// TIA Portal project "OI455" (V15.1)

(* hardware
DEVICE "ET 200SP station_1"  ET 200SP-Station
   slot 0: "Rack_0"  Rack  6ES5 710-8MAx1
   slot 1: "PLC_1"  CPU 1512SP-1 PN  6ES7 512-1DK01-0AB0  V2.6
   slot 2: "CM PtP_1"  CM PtP  6ES7 137-6AA00-0BA0  V1.0
      slot 1: "CM PtP_1"  CM PtP Sub
   slot 3: "CM PtP_2"  CM PtP  6ES7 137-6AA00-0BA0  V1.0
      slot 1: "CM PtP_2"  CM PtP Sub
   slot 4: "DI 8x24VDC BA_1"  DI 8x24VDC BA  6ES7 131-6BF01-0AA0  V0.0
      slot 1: "DI 8x24VDC BA_1"  DI 8x24VDC BA
   slot 5: "DI 8x24VDC BA_2"  DI 8x24VDC BA  6ES7 131-6BF01-0AA0  V0.0
      slot 1: "DI 8x24VDC BA_2"  DI 8x24VDC BA
   slot 6: "DI 8x24VDC BA_3"  DI 8x24VDC BA  6ES7 131-6BF01-0AA0  V0.0
      slot 1: "DI 8x24VDC BA_3"  DI 8x24VDC BA
   slot 7: "DQ 8x24VDC/0.5A BA_1"  DQ 8x24VDC/0.5A BA  6ES7 132-6BF01-0AA0  V0.0
      slot 1: "DQ 8x24VDC/0.5A BA_1"  DQ 8x24VDC/0.5A BA
   slot 8: "DQ 8x24VDC/0.5A BA_2"  DQ 8x24VDC/0.5A BA  6ES7 132-6BF01-0AA0  V0.0
      slot 1: "DQ 8x24VDC/0.5A BA_2"  DQ 8x24VDC/0.5A BA
   slot 9: "AI 8xI 2-,4-wire BA_1"  AI 8xI 2-,4-wire BA  6ES7 134-6GF00-0AA1  V1.0
      slot 1: "AI 8xI 2-,4-wire BA_1"  AI 8xI 2-,4-wire BA
   slot 10: "AI 8xI 2-,4-wire BA_2"  AI 8xI 2-,4-wire BA  6ES7 134-6GF00-0AA1  V1.0
      slot 1: "AI 8xI 2-,4-wire BA_2"  AI 8xI 2-,4-wire BA
   slot 11: "Server module_1"  Server module  6ES7 193-6PA00-0AA0  V1.1
      slot 1: "Server module_1"  Server module
   slot 127: "BA 2xRJ45"  BA 2xRJ45  6ES7 193-6AR00-0AA0  V0.0
      slot 32769: "Port_1"  6ES7 193-6AR00-0AA0
      slot 32770: "Port_2"  6ES7 193-6AR00-0AA0
*)

// ===== PLC "PLC_1"  CPU 1512SP-1 PN =====

VAR_GLOBAL   // PLC tag table "Default tag table"
   "AI2_Ch0" AT %IW35 : Word;
   "AI2_Ch1" AT %IW37 : Word;
   "AI2_Ch2" AT %IW39 : Word;
   "AI2_Ch3" AT %IW41 : Word;
   "AI2_Ch4" AT %IW43 : Word;
   "AI2_Ch5" AT %IW45 : Word;
   "AI2_Ch6" AT %IW47 : Word;
   "AI2_Ch7" AT %IW49 : Word;
   "AI1_Ch0" AT %IW19 : Word;
   "AI1_Ch1" AT %IW21 : Word;
   "AI1_Ch2" AT %IW23 : Word;
   "AI1_Ch3" AT %IW25 : Word;
   "AI1_Ch4" AT %IW27 : Word;
   "AI1_Ch5" AT %IW29 : Word;
   "AI1_Ch6" AT %IW31 : Word;
   "AI1_Ch7" AT %IW33 : Word;
   "DI1_In" AT %IB16 : Byte;
   "DI2_In" AT %IB17 : Byte;
   "DI3_In" AT %IB18 : Byte;
   "DO1_Out" AT %QB0 : Byte;
   "DO2_Out" AT %QB1 : Byte;
   "System_Byte" AT %MB1 : Byte;
   "FirstScan" AT %M1.0 : Bool;
   "DiagStatusUpdate" AT %M1.1 : Bool;
   "AlwaysTRUE" AT %M1.2 : Bool;
   "AlwaysFALSE" AT %M1.3 : Bool;
   "Clock_Byte" AT %MB0 : Byte;
   "Clock_10Hz" AT %M0.0 : Bool;
   "Clock_5Hz" AT %M0.1 : Bool;
   "Clock_2.5Hz" AT %M0.2 : Bool;
   "Clock_2Hz" AT %M0.3 : Bool;
   "Clock_1.25Hz" AT %M0.4 : Bool;
   "Clock_1Hz" AT %M0.5 : Bool;
   "Clock_0.625Hz" AT %M0.6 : Bool;
   "Clock_0.5Hz" AT %M0.7 : Bool;
   "ReqUVP" AT %M20.0 : Bool;
   "PrevState" AT %MW30 : Int;
   "HS600_active" AT %M20.1 : Bool;
   "Alarm_protect_XV100" AT %M20.2 : Bool;
   "Alarm_protect_XV100_prev" AT %M20.3 : Bool;
   "Alarm_Gas" AT %M20.4 : Bool;
   "Alarm_Gas_prev" AT %M20.5 : Bool;
   "Head_cmd_on_prev" AT %M20.6 : Bool;
   "Head_cmd_off_prev" AT %M20.7 : Bool;
   "Power_cmd_on_prev" AT %M21.0 : Bool;
   "Power_cmd_off_prev" AT %M21.1 : Bool;
   "CommandHMI_Spark_prev" AT %M21.2 : Bool;
   "Power_reset_prev" AT %M21.3 : Bool;
   "Head_reset_prev" AT %M21.4 : Bool;
END_VAR

TYPE "dt_AI"
   STRUCT
      Acp : DInt;   // Actual ADC code
      State : Word;
      Value : Real;   // Actual value (eng.units)
      Value_LastScan : Real;   // Last scan value
      K_filtr : Real := 0.0;   // Filter quoficient ( enable if K_filtr>0 )
      Circuit : Real;   // Actual current(mA)
      Voltage : Real;   // Actual vlotage (V)
      Resistance : Real;   // Input resistance (for voltage inputs)
      Scal_Max_Eu : Real := 100.0;   // Max scale value (eng.units)
      Scal_Min_Eu : Real := 0.0;   // Min scale value (eng.units)
      HH_Lim : Real := 100.0;   // HiHi alarm SP (eng.units)
      H_Lim : Real := 95.0;   // Hi warning SP (eng.units)
      L_Lim : Real := 5.0;   // Low warning SP (eng.units)
      LL_Lim : Real := 0.0;   // LowLow alarm SP (eng.units)
      HH_DeadBand : Real;   // HiHi alarm deadband
      H_DeadBand : Real;   // Hi warning deadband
      L_DeadBand : Real;   // Low warning deadband
      LL_DeadBand : Real;   // LowLow alarm deadband
      HH_Delay : Time;   // HiHi alarm SP delay
      H_Delay : Time;   // Hi warning SP delay
      L_Delay : Time;   // Low warning SP delay
      LL_Delay : Time;   // LowLow alarm SP delay
      Sim_Value : Real;   // Simulate value (eng.units)
      Sim_En : Bool := FALSE;   // Enable simulate mode
      Scal_Max_Upper : Bool;   // Flag Hi scale overflow
      Scal_Min_Under : Bool;   // Flag Low scale underflow
      Scale_0_20mA : Bool := FALSE;   // True - 0-20 mA, False - 4-20 mA
      Input_4mA_on_0_20mA : Bool := TRUE;   // True - 4-20mA sensor on 0-20mA current input
      VoltageInputType : Bool := FALSE;   // True -- voltage inpit, False - circuit input
      HH_Alarm : Bool;   // HiHi alarm flag
      H_Alarm : Bool;   // Hi warning flag
      L_Alarm : Bool;   // Low warning flag
      LL_Alarm : Bool;   // LowLow alarm flag
      HH_Alarm_En : Bool := TRUE;   // Enable HiHi alarm
      H_Alarm_En : Bool := FALSE;   // Enable Hi warning
      L_Alarm_En : Bool := FALSE;   // Enable Low warning
      LL_Alarm_En : Bool := TRUE;   // Enable LowLow alarm
      Short_Circuit : Bool;   // Shortcut flag
      Break : Bool;   // Breakoff flag
      Chan_Fail : Bool;   // Channel fault flag
      HH_Alarm_Logic : Bool;   // HiHi alarm for logic
      H_Alarm_Logic : Bool;   // Hi warning for logic
      L_Alarm_Logic : Bool;   // Low warning for logic
      LL_Alarm_Logic : Bool;   // LowLow alarm for logic
      Chan_Fail_Logic : Bool;   // Channel fault for logic
      Mask_mode : Bool;
      Test_mode : Bool;
      Ack_HH : Bool;
      Ack_H : Bool;
      Ack_L : Bool;
      Ack_LL : Bool;
      State_color : Byte;   // for HMI
      Ack_Alarm : Byte;   // for HMI
      Ack_Warning : Byte;   // for HMI
   END_STRUCT;
END_TYPE

TYPE "dt_DO"
   STRUCT
      Data_to_out : Word;
      Pins : Array[0..15] of Bool;
      UsePinsAsInput : Bool;
      Invert_En : Word;
      Output_En : Word;
      Sim_En : Word;
      Sim_Value : Word;
      Value : Word;
   END_STRUCT;
END_TYPE

TYPE "UVP_Param"
   STRUCT
      Connect_ID : UInt;
      IP_OCTET1 : UInt;
      IP_OCTET2 : UInt;
      IP_OCTET3 : UInt;
      IP_OCTET4 : UInt;
      IP_PORT : UInt;
   END_STRUCT;
END_TYPE

TYPE "Setpoints_v2"
   STRUCT
      UVPTimeCorrection : Real;
      reserv_4 : Real;
      reserv_5 : Real;
      reserv_6 : Real;
      Temp_L1_Press : Real;   // нижняя предупредительная уставка расхода газа на линии 2
      Temp_L1_Abs_Press : Real;
      Temp_L2_Press : Real;
      Temp_L2_Abs_Press : Real;
      Temp_L3_Press : Real;
      Temp_L3_Abs_Press : Real;
      Temp_L4_Press : Real;
      Temp_L4_Abs_Press : Real;
   END_STRUCT;
END_TYPE

TYPE "MeasuredUVP"
   STRUCT
      UVP_Press : Real;   // Избыточное давление, Па
      UVP_Abs_press : Real;   // Абсолютное давление, Па
      UVP_Temp : Real;   // Температура газа, С
      UVP_Ent : Real;   // Энтальпия, Дж/кг
      UVP_mass_flow : Real;   // Масовый расход, кг/сек
      UVP_Mass : Real;   // Масса, кг
      UVP_Vol_work : Real;   // Объем в р.у., м3
      UVP_Vol_norm : Real;   // Объем в ст.у., нм3
      UVP_T_power : Real;   // Тепловая мощность, Вт
      UVP_T_energ : Real;   // Тепловая энергия, Дж
      UVP_Time : DInt;   // Время штатной работы, сек
      UVP_TimeEr : DInt;   // Время нештатных ситуаций, сек
      UVP_Param_m_flow : Real;   // Параметр датчика расхода/количества, кг/сек
      UVP_Param_vol_flow_work : Real;   // Параметр датчика расхода/количества (в р.у.), м3/сек
      UVP_Param_vol_flow_norm : Real;   // Параметр датчика расхода/количества (в ст.у.), нм3/сек
      UVP_Param_mass : Real;   // Параметр датчика расхода/количества (масса), кг
      UVP_Param_vol : Real;   // Параметр датчика расхода/количества (объём в р.у.), м3
      UVP_NotUsed : Real;   // Резерв
      UVP_Density_norm : Real;   // Текущее значение плотности среды в ст.у, кг/м3
      UVP_Density_work : Real;   // Текущее значение плотности среды в р.у, кг/м3
      UVP_dP : Real;   // Перепад давления для трубопроводов на СУ, Па
      UVP_vol_flow_norm : Real;   // Объемный расход в ст.у. нм3/с
      UVP_vol_flow_work : Real;   // Объемный расход в р.у. нм3/с
   END_STRUCT;
END_TYPE

TYPE "CumulativeUVP"
   STRUCT
      UVP_Mass_prev2h : Real;   // Масса за предыд. час/2 часа, кг
      UVP_Vol_work_prev2h : Real;   // Объём в р.у за предыд. час/2 часа, м3
      UVP_Vol_norm_prev2h : Real;   // Объём в ст.у за предыд. час/2 часа, нм3
      UVP_Param_m_flow_prev2h : Real;   // Параметр датчика расхода/количества за предыд. час/2 часа, кг
      UVP_Param_vol_flow_work_prev2h : Real;   // Параметр датчика расхода/количества (объём в р.у.) за предыд. час/2 часа, м3
      UVP_Mass_cumul2h : Real;   // Масса на конец предыд. час/2 часа, кг
      UVP_Vol_work_cumul2h : Real;   // Объём на конец р.у за предыд. час/2 часа, м3
      UVP_Vol_norm_cumul2h : Real;   // Объём на конец ст.у за предыд. час/2 часа, нм3
      UVP_Param_m_flow_cumul2h : Real;   // Параметр датчика расхода/количества на конец предыд. час/2 часа, кг
      UVP_Param_vol_flow_work_cumul2h : Real;   // Параметр датчика расхода/количества (объём в р.у.) на конец предыд. час/2 часа, м3
      UVP_Mass_prevDay : Real;   // Масса за предыд. сутки, кг
      UVP_Vol_work_prevDay : Real;   // Объём в р.у за предыд. сутки, м3
      UVP_Vol_norm_prevDay : Real;   // Объём в ст.у за предыд. сутки, нм3
      UVP_Param_m_flow_prevDay : Real;   // Параметр датчика расхода/количества за предыд. сутки, кг
      UVP_Param_vol_flow_work_prevDay : Real;   // Параметр датчика расхода/количества (объём в р.у.) за предыд. сутки, м3
      UVP_Mass_cumulDay : Real;   // Масса на конец предыд. суток, кг
      UVP_Vol_work_cumulDay : Real;   // Объём на конец р.у за предыд. суток, м3
      UVP_Vol_norm_cumulDay : Real;   // Объём на конец ст.у за предыд. суток, нм3
      UVP_Param_m_flow_cumulDay : Real;   // Параметр датчика расхода/количества на конец предыд. суток, кг
      UVP_Param_vol_flow_work_cumulDay : Real;   // Параметр датчика расхода/количества (объём в р.у.) на конец предыд. суток, м3
   END_STRUCT;
END_TYPE

TYPE "Commands_v2"
   STRUCT
      Set_IP_UVP1 : Bool;   // Изменить IP адрес УВП1
      Set_IP_UVP2 : Bool;   // Изменить IP адрес УВП2
      UVP_MR113_Read : Bool;   // Прочитать компонентный состав из УВП 1
      UVP_MR113_Write : Bool;   // Записать компонентный состав в УВП 1
      UVP2_MR113_Read : Bool;   // Прочитать компонентный состав из УВП 2
      UVP2_MR113_Write : Bool;   // Записать компонентный состав в УВП 2
      UVPArchReadStart : Bool;   // команда на чтение архивной записи
   END_STRUCT;
END_TYPE

TYPE "DateTimeUVP"
   STRUCT
      Day : Int;
      Month : Int;
      Year : Int;
      Hour : Int;
      Minute : Int;
      Second : Int;
   END_STRUCT;
END_TYPE

TYPE "MR113_03_Gas_UVP"
   STRUCT
      CH4 : Real;   // Концентрация CH4 метан (мольные доли либо массовый %)
      C2H6 : Real;   // Концентрация C2H6 этан (мольные доли либо массовый %)
      C3H8 : Real;   // Концентрация C3H8 пропан (мольные доли либо массовый %)
      nC4H10 : Real;   // Концентрация н-C4H10 н-бутан (мольные доли либо массовый %)
      iC4H10 : Real;   // Концентрация и-C4H10 и-бутан (мольные доли либо массовый %)
      nC5H12 : Real;   // Концентрация н-C5H12 н-пептан (мольные доли либо массовый %)
      N2 : Real;   // Концентрация N2 азот (мольные доли либо массовый %)
      CO2 : Real;   // Концентрация CO2 углекислота (мольные доли либо массовый %)
      H2O : Real;   // Концентрация H2O вода (мольные доли либо массовый %)
      H2S : Real;   // Концентрация H2S сероводород (мольные доли либо массовый %)
      C6H14 : Real;   // Концентрация C6H14 гексан (мольные доли либо массовый %)
      C7H16 : Real;   // Концентрация C7H16 гептан (мольные доли либо массовый %)
      O2 : Real;   // Концентрация O2 кислород (мольные доли либо массовый %)
      iC5H12 : Real;   // Концентрация и-C5H12 и-пептан (мольные доли либо массовый %)
      Humidity : Real;   // Влажность (абсолютное значение в г/м3 либо относительная концентрация)
   END_STRUCT;
END_TYPE

TYPE "Measured"
   STRUCT
      UVP1_L1_Archive_AbsPresAve : Real;   // Архивное давление, МПа (среднее за период) - УВП1 линия1
      UVP1_L1_Archive_AbsTempAve : Real;   // Архивная температура, С (средняя за период) - УВП1 линия1
      UVP1_L1_Archive_FlowWorkPeriod : Real := 0.0;   // Архивный расход за период (р.у.), м3 - УВП1 линия1
      UVP1_L1_Archive_FlowNormPeriod : Real := 0.0;   // Архивный расход за период (с.у.), нм3 - УВП1 линия1
      UVP1_L1_Archive_StableWorkTime : Real := 0.0;   // Время штатной работы, часов - УВП1 линия1
      reserv : Real := 0.0;   // резерв
      UVP1_L2_Archive_AbsPresAve : Real := 0.0;   // Архивное давление, МПа (среднее за период) - УВП1 линия2
      UVP1_L2_Archive_AbsTempAve : Real := 0.0;   // Архивная температура, С (средняя за период) - УВП1 линия2
      UVP1_L2_Archive_FlowWorkPeriod : Real := 0.0;   // Архивный расход за период (р.у.), м3 - УВП1 линия2
      UVP1_L2_Archive_FlowNormPeriod : Real := 0.0;   // Архивный расход за период (с.у.), нм3 - УВП1 линия2
      UVP1_L2_Archive_StableWorkTime : Real := 0.0;   // Время штатной работы, часов - УВП1 линия2
      reserv_6 : Real := 0.0;   // резерв
      UVP1_L3_Archive_AbsPresAve : Real := 0.0;   // Архивное давление, МПа (среднее за период) - УВП1 линия3
      UVP1_L3_Archive_AbsTempAve : Real := 0.0;   // Архивная температура, С (средняя за период) - УВП1 линия3
      UVP1_L3_Archive_FlowWorkPeriod : Real := 0.0;   // Архивный расход за период (р.у.), м3 - УВП1 линия3
      UVP1_L3_Archive_FlowNormPeriod : Real := 0.0;   // Архивный расход за период (с.у.), нм3 - УВП1 линия3
      UVP1_L3_Archive_StableWorkTime : Real := 0.0;   // Время штатной работы, часов - УВП1 линия3
      reserv_12 : Real := 0.0;   // резерв
      UVP1_L4_Archive_AbsPresAve : Real;   // Архивное давление, МПа (среднее за период) - УВП1 линия4
      UVP1_L4_Archive_AbsTempAve : Real;   // Архивная температура, С (средняя за период) - УВП1 линия4
      UVP1_L4_Archive_FlowWorkPeriod : Real;   // Архивный расход за период (р.у.), м3 - УВП1 линия4
      UVP1_L4_Archive_FlowNormPeriod : Real;   // Архивный расход за период (с.у.), нм3 - УВП1 линия4
      UVP1_L4_Archive_StableWorkTime : Real;   // Время штатной работы, часов - УВП1 линия4
      reserv_18 : Real;   // резерв
      UVP2_L1_Archive_AbsPresAve : Real;   // Архивное давление, МПа (среднее за период) - УВП1 линия1
      UVP2_L1_Archive_AbsTempAve : Real;   // Архивная температура, С (средняя за период) - УВП2 линия1
      UVP2_L1_Archive_FlowWorkPeriod : Real := 0.0;   // Архивный расход за период (р.у.), м3 - УВП2 линия1
      UVP2_L1_Archive_FlowNormPeriod : Real := 0.0;   // Архивный расход за период (с.у.), нм3 - УВП2 линия1
      UVP2_L1_Archive_StableWorkTime : Real := 0.0;   // Время штатной работы, часов - УВП2 линия1
      reserv_1 : Real := 0.0;   // резерв
      UVP2_L2_Archive_AbsPresAve : Real := 0.0;   // Архивное давление, МПа (среднее за период) - УВП2 линия2
      UVP2_L2_Archive_AbsTempAve : Real := 0.0;   // Архивная температура, С (средняя за период) - УВП2 линия2
      UVP2_L2_Archive_FlowWorkPeriod : Real := 0.0;   // Архивный расход за период (р.у.), м3 - УВП2 линия2
      UVP2_L2_Archive_FlowNormPeriod : Real := 0.0;   // Архивный расход за период (с.у.), нм3 - УВП2 линия2
      UVP2_L2_Archive_StableWorkTime : Real := 0.0;   // Время штатной работы, часов - УВП2 линия2
      reserv_7 : Real := 0.0;   // резерв
      reserv_19 : Real;   // резерв
   END_STRUCT;
END_TYPE

TYPE "MR113_03_Gas_UVP_Int"
   STRUCT
      Concentration : Int;
      Water : Int;
   END_STRUCT;
END_TYPE

TYPE "UVP_ArchiveResult"
   STRUCT
      UVP1_Archive_RequestStatus : Int;   // Статус чтения архива (для первого клиента): 0 - нет данных, 1 - идёт сбор, 2 - данные готовы, 3..7 - ошибки
      UVP2_Archive_RequestStatus : Int;   // Статус чтения архива (для второго клиента): 0 - нет данных, 1 - идёт сбор, 2 - данные готовы, 3..7 - ошибки
      UVP3_Archive_RequestStatus : Int;   // Статус чтения архива (для третьего клиента): 0 - нет данных, 1 - идёт сбор, 2 - данные готовы, 3..7 - ошибки
      UVP4_Archive_RequestStatus : Int;   // резерв
      UVP1_Archive_Update_Data : Int;
      UVP2_Archive_Update_Data : Int;
      UVP3_Archive_Update_Data : Int;
      UVP4_Archive_Update_Data : Int;
      reserv : Int;
      reserv_1 : Int;
      reserv_2 : Int;
      reserv_3 : Int;
      reserv_4 : Int;
      reserv_5 : Int;
      reserv_6 : Int;
      reserv_7 : Int;
      reserv_8 : Int;
      reserv_9 : Int;
   END_STRUCT;
END_TYPE

TYPE "Flags_v2"
   STRUCT
      UVP1_main : Bool := FALSE;   // Выбран УВП 1
      UVP2_main : Bool := FALSE;   // Выбран УВП 2
      UVP1_on : Bool := FALSE;   // Наличие связи с УВП1
      UVP2_on : Bool := FALSE;   // Наличие связи с УВП2
      NonCorPrimDate : Bool := FALSE;   // Ошибка в начальном времени запроса архивных данных
      NonCorFinDate : Bool := FALSE;   // Ошибка в конечном времени запроса архивных данных
      NonCorNumLine : Bool;   // Ошибка в задании номера трубопровода
      LargePeriod : Bool;   // Слишком большой период для сбора данных
      RezNonValid : Bool;   // Резу-т запроса уничтожен по таймауту или запрос не был воспринят УВП
      NonNote : Bool;   // За выбранный период в архиве нет ни одной записи
   END_STRUCT;
END_TYPE

TYPE "UVP_Param_1"
   STRUCT
      Connect_ID : UInt;
      IP_OCTET1 : Byte;
      IP_OCTET2 : Byte;
      IP_OCTET3 : Byte;
      IP_OCTET4 : Byte;
      IP_PORT : UInt;
   END_STRUCT;
END_TYPE

TYPE "ClientMode"
   STRUCT
      Mode : USInt;
      Data_ADDR : UDInt;
      Data_LEN : UInt;
   END_STRUCT;
END_TYPE

TYPE "Client"
   STRUCT
      Done : Bool;
      Busy : Bool;
      Error : Bool;
      Status : Word;
      Disconnect : Bool;
   END_STRUCT;
END_TYPE

TYPE "REG_State"
   STRUCT
      Open : Bool;
      Close : Bool;
      Mufta_on_open : Bool;
      Mufta_on_close : Bool;
      res : Bool;
      Battery_low : Bool;
      res_1 : Bool;
      DU_MU : Bool;
      Openning : Bool;
      Closing : Bool;
      Stoping : Bool;
      Sboi_DP : Bool;
      Work_on_AI : Bool;
      Warm_on : Bool;
      AI_input_outoff_range : Bool;
      Ready : Bool;
   END_STRUCT;
END_TYPE

TYPE "REG_Defects"
   STRUCT
      reserv : Bool;
      Def2_on : Bool;
      Def8_on : Bool;
      Def6_on : Bool;
      Def12_on : Bool;
      Def23_on : Bool;
      Def19_on : Bool;
      Def5_on : Bool;
      Def13_on : Bool;
      Def22_on : Bool;
      Def7_on : Bool;
      Def3_on : Bool;
      Def4_on : Bool;
      Def11_on : Bool;
      Def15_on : Bool;
      Def16_on : Bool;
   END_STRUCT;
END_TYPE

TYPE "REG_Commands"
   STRUCT
      Stop : Bool;
      Open : Bool;
      Close : Bool;
      res_3 : Bool;
      res_4 : Bool;
      Reset : Bool;
      res_5 : Bool;
      res_6 : Bool;
      res_7 : Bool;
      res_8 : Bool;
      res_9 : Bool;
      res_10 : Bool;
      res_11 : Bool;
      res_12 : Bool;
      res_13 : Bool;
      res_14 : Bool;
   END_STRUCT;
END_TYPE

TYPE "MasterSetttings"
   STRUCT
      MB_Addr : UInt;
      Done : Bool;
      Busy : Bool;
      Error : Bool;
      Status : Word;
   END_STRUCT;
END_TYPE

TYPE "MasterMode"
   STRUCT
      Mode : USInt;
      Data_Addr : UDInt;
      Data_Len : UInt;
   END_STRUCT;
END_TYPE

TYPE "AUMA_Message"
   STRUCT
      End_position_OPEN : Bool;
      End_position_CLOSE : Bool;
      LOSS_end_position : Bool;
      No_ready_DIST : Bool;
      OPENING : Bool;
      CLOSING : Bool;
      Warning : Bool;
      Error : Bool;
      Term_error : Bool;
      Phase_failure : Bool;
      Selector_DIST : Bool;
      Selector_LOCAL : Bool;
      Limit_switch_OPEN : Bool;
      Limit_switch_CLOSE : Bool;
      Moment_switch_OPEN : Bool;
      Moment_switch_CLOSE : Bool;
   END_STRUCT;
END_TYPE

TYPE "AUMA_Status"
   STRUCT
      No_ready_DIST : Bool;
      Warning : Bool;
      Error : Bool;
      Maintenance : Bool;
      Out_specification : Bool;
      Function_check : Bool;
      Fail : Bool;
      Device_normal : Bool;
      Pause_movement : Bool;
      Intermediate_position : Bool;
      Step_mode : Bool;
      rezerv : Bool;
      Drive_running : Bool;
      Flywheel_travel : Bool;
      Moving_DU : Bool;
      Moving_LOCAL : Bool;
   END_STRUCT;
END_TYPE

TYPE "PortConfig"
   STRUCT
      Port : Port;
      Baud : UDInt;
      Parity : UInt;
      Done : Bool;
      Error : Bool;
      Status : Word;
      test : Int;
   END_STRUCT;
END_TYPE

TYPE "Command"
   STRUCT
      Control_line : UInt;   // 0-нет команды,1-налив,2-стоп,3-сброс,4-пауза,5-продолжить
      Dose : UDInt;   // Доза отпуска (кг/л)
      Unit_code : UInt;   // Код единицы отпуска (0-кг,1-литры)
      Device_choice : UInt;   // Схема процеса (0-верхний налив,1-нижний)
      Mode : UInt;   // Режим работы (0-стд,1-расш отображ,2-отладка,3,4-тест)
      Reserv : UInt;   // резерв
      Porog_min_to_max : UInt;   // Порог перехода с мин расхода на макс в нач замера
      Porog_max_to_min : UInt;   // Порог перехода с макс расхода на мин в нач замера
      Control_line_enable : UInt;   // Разрешение команды упр-я АСН от АРМ (бит00-налив,01-стоп,02-пауза,03-продожить,04-подтв/сброс)
   END_STRUCT;
END_TYPE

TYPE "State_line"
   STRUCT
      Curr_operations : Struct   // Текущие показатели
         P_izb_oil : Real;   // Изб.давление, МПа
         T_oil : Real;   // Температура продукта, С
         P_oil : Real;   // Плотность продукта, кг/м3
         Duration_min : UInt;   // Длит тек операции налива, мин
         Duration_sec : UInt;   // Длит тек операции налива, сек
         res_0 : UInt;
         res_1 : UInt;
         Sum_M_brut : UDInt;   // Сум.накопл.продукт, масса бруто, кг
         F_oil_brut : Real;   // Расход продукта брутто масс., кг/ч
         D_oil_net : Real;   // Расход продукта нетто масс., кг/ч
         D_wtr : Real;   // Дебит воды масс, кг/ч
         Watercut_M : Real;   // Обводненность массовая, кг/кг %
         Sum_vol_wrk : UDInt;   // Сумм.накопл.продукт,объем брутто в раб.усл., л
         D_oil_V_brut_wrk : Real;   // Дебит продукта брутто объемный в раб.усл., л/ч
         D_oil_V_nett_wrk : Real;   // Дебит продукта нетто объемный в раб.усл., л/ч
         D_wtr_V_wrk : Real;   // Дебит воды объемный в раб.усл., л/ч
         Watercut_V_wrk : Real;   // Обводненность жидкости объем. в раб.усл., л/л %
         Sum_V_brut_std : UDInt;   // Сумм.накопл.продукт,объем брутто в ст.усл., л
         D_oil_V_brut_std : Real;   // Дебит продукта брутто объемный в ст.усл., л/ч
         D_oil_V_nett_std : Real;   // Дебит продукта нетто объемный в ст.усл., л/ч
         D_wtr_V_std : Real;   // Дебит воды объемный в ст.усл., л/ч
         Watercut_V_std : Real;   // Обводненность жидкости объем. в ст.усл., л/л %
      END_STRUCT;
      Aver_operations : Struct   // Усредненные показатели
         P_izb_oil : Real;   // Изб.давление, МПа
         T_oil : Real;   // Температура продукта, С
         P_oil : Real;   // Плотность продукта, кг/м3
         Duration_min : UInt;   // Длит тек операции налива, мин
         Duration_sec : UInt;   // Длит тек операции налива, сек
         res_0 : UInt;
         res_1 : UInt;
         Sum_M_brut : UDInt;   // Сум.накопл.продукт, масса бруто, кг
         F_oil_brut : Real;   // Расход продукта брутто масс., кг/ч
         D_oil_net : Real;   // Расход продукта нетто масс., кг/ч
         D_wtr_1 : Real;   // Дебит воды масс, кг/ч
         Watercut_M : Real;   // Обводненность массовая, кг/кг %
         Sum_vol_wrk : UDInt;   // Сумм.накопл.продукт,объем брутто в раб.усл., л
         D_oil_V_brut_wrk : Real;   // Дебит продукта брутто объемный в раб.усл., л/ч
         D_oil_V_nett_wrk : Real;   // Дебит продукта нетто объемный в раб.усл., л/ч
         D_wtr_V_wrk : Real;   // Дебит воды объемный в раб.усл., л/ч
         Watercut_V_wrk : Real;   // Обводненность жидкости объем. в раб.усл., л/л %
         Sum_V_brut_std : UInt;   // Сумм.накопл.продукт,объем брутто в ст.усл., л
         D_oil_V_brut_std : Real;   // Дебит продукта брутто объемный в ст.усл., л/ч
         D_oil_V_nett_std : Real;   // Дебит продукта нетто объемный в ст.усл., л/ч
         D_wtr_V_std : Real;   // Дебит воды объемный в ст.усл., л/ч
         Watercut_V_std : Real;   // Обводненность жидкости объем. в ст.усл., л/л %
         Sum_mass : Real;   // Сумм накопл.продукт, масса брутто, кг
         Sum_vol : Real;   // Сумм накопл.продукт, объем брутто, л
         Sum_mass_all : LReal;   // Сумм накопл.продукт, масса брутто, кг (несбрас)
         Sum_vol_all : LReal;   // Сумм накопл.продукт, объем брутто, л (несбрас)
      END_STRUCT;
   END_STRUCT;
END_TYPE

TYPE "Command_sec"
   STRUCT
      Control_line : UInt;   // 0-нет команды,1-налив,2-стоп,3-сброс,4-пауза,5-продолжить
      Dose : UDInt;   // Доза отпуска (кг/л)
      Unit_code : UInt;   // Код единицы отпуска (0-кг,1-литры)
      Device_choice : UInt;   // Схема процеса (0-верхний налив,1-нижний)
      Mode : UInt;   // Режим работы (0-стд,1-расш отображ,2-отладка,3,4-тест)
      Reserv : UInt;   // резерв
      Porog_min_to_max : UInt;   // Порог перехода с мин расхода на макс в нач замера
      Porog_max_to_min : UInt;   // Порог перехода с макс расхода на мин в нач замера
   END_STRUCT;
END_TYPE

DATA_BLOCK "Head"   // DB31
{ S7_Optimized_Access := 'FALSE' }
NAME : Scan_Dev
VERSION : 1.2
// stored: InstanceOfName Scan_Dev
"Scan_Dev"
BEGIN
END_DATA_BLOCK

DATA_BLOCK "Power"   // DB32
{ S7_Optimized_Access := 'FALSE' }
NAME : Scan_Dev
VERSION : 1.2
// stored: InstanceOfName Scan_Dev
"Scan_Dev"
BEGIN
END_DATA_BLOCK

// folder: AI_DB

DATA_BLOCK "PT100"   // DB1
{ S7_Optimized_Access := 'FALSE' }
NAME : Scan_AI
VERSION : 1.3
// stored: InstanceOfName Scan_AI
"Scan_AI"
BEGIN
END_DATA_BLOCK

DATA_BLOCK "TT100"   // DB2
{ S7_Optimized_Access := 'FALSE' }
NAME : Scan_AI
VERSION : 1.3
// stored: InstanceOfName Scan_AI
"Scan_AI"
BEGIN
END_DATA_BLOCK

DATA_BLOCK "LT100"   // DB3
{ S7_Optimized_Access := 'FALSE' }
NAME : Scan_AI
VERSION : 1.3
// stored: InstanceOfName Scan_AI
"Scan_AI"
BEGIN
END_DATA_BLOCK

DATA_BLOCK "AG100"   // DB4
{ S7_Optimized_Access := 'FALSE' }
NAME : Scan_AI
VERSION : 1.3
// stored: InstanceOfName Scan_AI
"Scan_AI"
BEGIN
END_DATA_BLOCK

DATA_BLOCK "PT200"   // DB5
{ S7_Optimized_Access := 'FALSE' }
NAME : Scan_AI
VERSION : 1.3
// stored: InstanceOfName Scan_AI
"Scan_AI"
BEGIN
END_DATA_BLOCK

DATA_BLOCK "TT200"   // DB6
{ S7_Optimized_Access := 'FALSE' }
NAME : Scan_AI
VERSION : 1.3
// stored: InstanceOfName Scan_AI
"Scan_AI"
BEGIN
END_DATA_BLOCK

DATA_BLOCK "LT200"   // DB7
{ S7_Optimized_Access := 'FALSE' }
NAME : Scan_AI
VERSION : 1.3
// stored: InstanceOfName Scan_AI
"Scan_AI"
BEGIN
END_DATA_BLOCK

DATA_BLOCK "AG200"   // DB8
{ S7_Optimized_Access := 'FALSE' }
NAME : Scan_AI
VERSION : 1.3
// stored: InstanceOfName Scan_AI
"Scan_AI"
BEGIN
END_DATA_BLOCK

DATA_BLOCK "TT500"   // DB9
{ S7_Optimized_Access := 'FALSE' }
NAME : Scan_AI
VERSION : 1.3
// stored: InstanceOfName Scan_AI
"Scan_AI"
BEGIN
END_DATA_BLOCK

// folder: DI_DO_DB

DATA_BLOCK "DI1"   // DB10
{ S7_Optimized_Access := 'TRUE' }
NAME : ScanDI08
VERSION : 1.2
// stored: InstanceOfName Scan_DI08
"Scan_DI08"
BEGIN
END_DATA_BLOCK

DATA_BLOCK "DI2"   // DB11
{ S7_Optimized_Access := 'TRUE' }
NAME : ScanDI08
VERSION : 1.2
// stored: InstanceOfName Scan_DI08
"Scan_DI08"
BEGIN
END_DATA_BLOCK

DATA_BLOCK "DI3"   // DB12
{ S7_Optimized_Access := 'TRUE' }
NAME : ScanDI08
VERSION : 1.2
// stored: InstanceOfName Scan_DI08
"Scan_DI08"
BEGIN
END_DATA_BLOCK

DATA_BLOCK "DO1"   // DB24
{ S7_Optimized_Access := 'TRUE' }
NAME : PutDO08
VERSION : 1.0
// stored: InstanceOfName Put_DO08
"Put_DO08"
BEGIN
END_DATA_BLOCK

DATA_BLOCK "DO2"   // DB25
{ S7_Optimized_Access := 'TRUE' }
NAME : PutDO08
VERSION : 1.0
// stored: InstanceOfName Put_DO08
"Put_DO08"
BEGIN
END_DATA_BLOCK

// folder: Modbus

DATA_BLOCK "UVP_Data"   // DB13
{ S7_Optimized_Access := 'FALSE' }
VERSION : 0.1
   VAR
      UVP1_Settings : "UVP_Param";   // Параметры подключения к УВП1
      Commands : "Commands_v2";   // Команды
      Setpoints : "Setpoints_v2";   // Уставки,пределы и т. д.
      Flags : "Flags_v2";   // Флаги
      UVP1_Current_L1 : "MeasuredUVP";   // Текущие параметры УВП (линия 1)
      UVP1_Cumulative_L1 : "CumulativeUVP";   // Накопительные параметры УВП (линия 1)
      UVP1_Current_L2 : "MeasuredUVP";   // Текущие параметры УВП (линия 2)
      UVP1_Cumulative_L2 : "CumulativeUVP";   // Накопительные параметры УВП (линия 2)
      UVP1_Current_L3 : "MeasuredUVP";   // Текущие параметры УВП (линия 3)
      UVP1_Cumulative_L3 : "CumulativeUVP";   // Накопительные параметры УВП (линия 3)
      UVP1_Current_L4 : "MeasuredUVP";   // Текущие параметры УВП (линия 4)
      UVP1_Cumulative_L4 : "CumulativeUVP";   // Накопительные параметры УВП (линия 4)
      UVP1_Current_L5 : "MeasuredUVP";   // Текущие параметры УВП (линия 5)
      UVP1_Cumulative_L5 : "CumulativeUVP";   // Накопительные параметры УВП (линия 5)
      UVP1_DateTime : "DateTimeUVP";   // Текущее время УВП
      UVP1_MR113 : "MR113_03_Gas_UVP";   // Компонентный состав газовой смеси МР113
      UVP1_MR113_Int : "MR113_03_Gas_UVP_Int";   // Компонентный состав газовой смеси МР113 (продолжение)
      UVP1_Archives : Struct   // Дата-время и номер т/п в запросе архива
         UVP_param : Int;
         UVP_line : Int;   // Начальная дата отчета: Номер трубопровода
         UVP_day : Int;   // Начальная дата отчета: 24
         UVP_month : Int;   // Начальная дата отчета: 6
         UVP_year : Int;   // Начальная дата отчета: В формате: "14" - значит 2014 год
         UVP_hour : Int;   // Начальная дата отчета: 6
         UVP_min : Int;   // Начальная дата отчета: 23
         UVP_sec : Int;   // Начальная дата отчета: 14
         UVP_day_end : Int;   // Конченая дата: 24
         UVP_month_end : Int;   // Конченая дата: 6
         UVP_year_end : Int;   // Конченая дата: 14
         UVP_hour_end : Int;   // Конченая дата: 6
         UVP_min_end : Int;   // Конченая дата:12
         UVP_sec_end : Int;   // Конченая дата: 15
      END_STRUCT;
      Archive_Results : "UVP_ArchiveResult";   // Ход и результаты чтения архивов выбранного УВП
      ArchiveData : "Measured";   // Архивные данные с УВП 1 и с УВП 2 обработанные!
      UVP1_Data_Arch : Array[0..7] of String[20];
      _terminator : Bool;   // завершающий элемент, для удобства вычисления длины блока
   END_VAR
BEGIN
   UVP1_Settings.Connect_ID := 1;
   UVP1_Settings.IP_OCTET1 := 192;
   UVP1_Settings.IP_OCTET2 := 168;
   UVP1_Settings.IP_OCTET4 := 170;
   UVP1_Settings.IP_PORT := 502;
END_DATA_BLOCK

DATA_BLOCK "UVP_States"   // DB14
{ S7_Optimized_Access := 'FALSE' }
VERSION : 0.1
   VAR
      Client : "Client";
      ReqReadOpData : "ClientMode";
      ReqWriteCom : "ClientMode";
      ReqReadArcData : "ClientMode";
      ReqReadAns : "ClientMode";
      ClientMode : "ClientMode";
      State : Int;
      NewState : Bool;
      Answer : Word;
      Data_PTR : Array[0..119] of Word;
      ArcDataString : String;
      SubString : Array[0..10] of String;
      ArcDataStOp : String;
      Format : Word;
      ArcData2 : Array[0..10] of String;
      UVP_Param : "UVP_Param_1";   // Текущие параметры для текущего УВП
      ReqReadOpData_dest_offset : Int;
      ReqReadOpData_nextState : Int;
      ArhDataParsed : Array[0..2, 0..10] of Real;
      ArchClientIndex : Int;   // Номер клиента (1..3), для которого сейчас вынимается архив из УВП
      SubStringT : Array[0..2, 0..1] of String[18];
      Connect_UVP : TCON_IP_v4;
   END_VAR
BEGIN
   Connect_UVP.ID := 16#0001;
   Connect_UVP.RemoteAddress.ADDR[1] := 192;
   Connect_UVP.RemoteAddress.ADDR[2] := 168;
   Connect_UVP.RemoteAddress.ADDR[3] := 0;
   Connect_UVP.RemoteAddress.ADDR[4] := 2;
   UVP_Param.Connect_ID := 1;
   UVP_Param.IP_OCTET1 := 192;
   UVP_Param.IP_OCTET2 := 168;
   UVP_Param.IP_OCTET3 := 0;
   UVP_Param.IP_OCTET4 := 2;
   UVP_Param.IP_PORT := 502;
END_DATA_BLOCK

DATA_BLOCK "REG_Data"   // DB15
{ S7_Optimized_Access := 'FALSE' }
VERSION : 0.1
   VAR
      reserv : Word;
      PCV300_Message : "AUMA_Message";
      PCV300_Pologenie : Int;
      PCV300_Status : "AUMA_Status";
      PCV300_Pologenie_ok : Real;
      PCV300_Setpoint : Int;
      LCV300_Message : "AUMA_Message";
      LCV300_Pologenie : Int;
      LCV300_Status : "AUMA_Status";
      LCV300_Pologenie_ok : Real;
      LCV300_Setpoint : Int;
   END_VAR
BEGIN
END_DATA_BLOCK

DATA_BLOCK "REG_Master"   // DB16
{ S7_Optimized_Access := 'FALSE' }
VERSION : 0.1
   VAR
      Settings : "MasterSetttings";
      Data : Array[0..10] of Word;
      State : Int;
      Data_offset : Int;
      DataAddrCommand : UDInt;
      MasterMode : "MasterMode";
      Next_State : Int;
      Prev_State : Int;
      Register : Int;
      reqREGmaster : Bool;
      PCV300_error : Bool;
      LCV300_error : Bool;
      reg_PCV300_err : Bool;   // Потеря связи с регулятором PCV300
      reg_LCV300_err : Bool;   // Потеря связи с регулятором LCV300
      count_PCV300 : Int;   // Счетчик пропуска циклов PCV300
      count_LCV300 : Int;   // Счетчик пропуска циклов LCV300
      PCV300_done_count : Int;
      LCV300_done_count : Int;
      test1 : Int;
   END_VAR
BEGIN
END_DATA_BLOCK

DATA_BLOCK "Regs"   // DB19
{ S7_Optimized_Access := 'TRUE' }
VERSION : 0.1
   VAR
      PCV300_Alarm : Bool;
      PCV300_Warning : Bool;
      PCV300_Remont : Bool;
      LCV300_Alarm : Bool;
      LCV300_Warning : Bool;
      LCV300_Remont : Bool;
      PCV300_Midle : Bool;
      LCV300_Midle : Bool;
   END_VAR
   VAR RETAIN
      PCV300_Man_En : Bool;
      LCV300_Man_En : Bool;
      PCV300_SP : Real;
      LCV300_SP : Real;
      PCV300_Man_Value : Real;
      LCV300_Man_Value : Real;
      PCV300_OutputUpperLimit : Real;
      LCV300_OutputUpperLimit : Real;
      PCV300_OutputLowerLimit : Real;
      LCV300_OutputLowerLimit : Real;
   END_VAR
BEGIN
END_DATA_BLOCK

DATA_BLOCK "PortSettings"   // DB21
{ S7_Optimized_Access := 'FALSE' }
VERSION : 0.1
   VAR
      Regs : "PortConfig";
      Up : "PortConfig";
      Slave_Up_NDR : Bool;
      Slave_Up_DR : Bool;
      Slave_Up_ERROR : Bool;
      Slave_Up_STATUS : Word;
   END_VAR
BEGIN
END_DATA_BLOCK

DATA_BLOCK "DATA"   // DB23
{ S7_Optimized_Access := 'FALSE' }
VERSION : 0.1
   VAR
      offset : Int;
      Measuring : Struct
         PT100_Value : Real;   // PT100_Значение
         PT100_Circuit : Real;   // PT100_Ток
         TT100_Value : Real;   // TT100_Значение
         TT100_Circuit : Real;   // TT100_Ток
         LT100_Value : Real;   // LT100_Значение
         LT100_Circuit : Real;   // LT100_Ток
         AG100_Value : Real;   // AG100_Значение
         AG100_Circuit : Real;   // AG100_Ток
         PT200_Value : Real;   // PT200_Значение
         PT200_Circuit : Real;   // PT200_Ток
         TT200_Value : Real;   // TT200_Значение
         TT200_Circuit : Real;   // TT200_Ток
         LT200_Value : Real;   // LT200_Значение
         LT200_Circuit : Real;   // LT200_Ток
         AG200_Value : Real;   // AG200_Значение
         AG200_Circuit : Real;   // AG200_Ток
         TT500_Value : Real;   // TT500_Значение
         TT500_Circuit : Real;   // TT500_Ток
         PCV300_Pologenie : Real;   // PCV300 Положение
         LCV300_Pologenie : Real;   // LCV300 Положение
         SIKG_Press : Real;   // Давление СИКГ
         SIKG_Temp : Real;   // Температура СИКГ
         SIKG_Flow_ru : Real;   // Расход (раб. усл.) СИКГ
         SIKG_Flow_stu : Real;   // Расход (ст. усл.) СИКГ
         SIKG_Flow_ru_prev2h : Real;   // Расход (раб. усл.) СИКГ за предыдущие 2 часа
         SIKG_Flow_stu_prev2h : Real;   // Расход (ст. усл.) СИКГ за предыдущие 2 часа
         SIKG_Flow_ru_prevDay : Real;   // Расход (раб. усл.) СИКГ за предыдущие сутки
         SIKG_Flow_stu_prevDay : Real;   // Расход (ст. усл.) СИКГ за предыдущие сутки
         SIKG_total : Real;   // Интегральный счетчик
         SIKN_MassFlow : Real;   // Массовый расход СИКН
         SIKN_MassFlow_prev2h : Real;   // Массовый расход СИКН за предыдущие 2 часа
         SIKN_MassFlow_prevDay : Real;   // Массовый расход СИКН за предыдущие сутки
         SIKN_total : Real;   // Интегральный счетчик
         XV100_State : Int;   // Состояние XV100: 0-неопределено, 1-закрыт, 2-открыт, 3-авария
         Head_State : Int;   // Состояние обогрева: 0-выключен, 1-включен, 2-авария
         Power_State : Int;   // Состояние питания: 0-выключен, 1-включен, 2-авария
         PCV300_Alarm : Bool;   // PCV300 авария
         PCV300_Warning : Bool;   // PCV300 предупреждение
         PCV300_Midle : Bool;   // PCV300 среднее положение
         PCV300_DIST : Bool;   // PCV300 дистанц. режим
         PCV300_LOCAL : Bool;   // PCV300 местный. режим
         LCV300_Alarm : Bool;   // LCV300 авария
         LCV300_Warning : Bool;   // LCV300 предупреждение
         LCV300_Midle : Bool;   // LCV300 среднее положение
         LCV300_DIST : Bool;   // LCV300 дистанц. режим
         LCV300_LOCAL : Bool;   // LCV300 местный. режим
         LS100 : Bool;   // LS100
         LS101 : Bool;   // LS101
         LS200 : Bool;   // LS200
         LS201 : Bool;   // LS201
         HS600_Emer_stop : Bool;   // Кнопка аварийного останова
         Head_run : Bool;   // Обогрев включен (сигнал с контактора)
         Power_run : Bool;   // Питание включено (сигнал с контактора)
         XV100_open : Bool;   // XV100 открыт (сигнал с задвижки)
         XV100_close : Bool;   // XV100 закрыт (сигнал с задвижки)
         XV100_fault : Bool;   // XV100 неисправность (сигнал с задвижки)
         XV100_no_cmd_close : Bool;   // XV100 не закрылся по команде
         XV100_no_cmd_open : Bool;   // XV100 не открылсяпо команде
         Spark : Bool;
         PT100_HH_Alarm : Bool;
         PT100_H_Alarm : Bool;
         PT100_L_Alarm : Bool;
         PT100_LL_Alarm : Bool;
         PT100_Chan_Fail : Bool;
         PT100_Sim : Bool;
         TT100_HH_Alarm : Bool;
         TT100_H_Alarm : Bool;
         TT100_L_Alarm : Bool;
         TT100_LL_Alarm : Bool;
         TT100_Chan_Fail : Bool;
         TT100_Sim : Bool;
         LT100_HH_Alarm : Bool;
         LT100_H_Alarm : Bool;
         LT100_L_Alarm : Bool;
         LT100_LL_Alarm : Bool;
         LT100_Chan_Fail : Bool;
         LT100_Sim : Bool;
         AG100_HH_Alarm : Bool;
         AG100_H_Alarm : Bool;
         AG100_L_Alarm : Bool;
         AG100_LL_Alarm : Bool;
         AG100_Chan_Fail : Bool;
         AG100_Sim : Bool;
         PT200_HH_Alarm : Bool;
         PT200_H_Alarm : Bool;
         PT200_L_Alarm : Bool;
         PT200_LL_Alarm : Bool;
         PT200_Chan_Fail : Bool;
         PT200_Sim : Bool;
         TT200_HH_Alarm : Bool;
         TT200_H_Alarm : Bool;
         TT200_L_Alarm : Bool;
         TT200_LL_Alarm : Bool;
         TT200_Chan_Fail : Bool;
         TT200_Sim : Bool;
         LT200_HH_Alarm : Bool;
         LT200_H_Alarm : Bool;
         LT200_L_Alarm : Bool;
         LT200_LL_Alarm : Bool;
         LT200_Chan_Fail : Bool;
         LT200_Sim : Bool;
         AG200_HH_Alarm : Bool;
         AG200_H_Alarm : Bool;
         AG200_L_Alarm : Bool;
         AG200_LL_Alarm : Bool;
         AG200_Chan_Fail : Bool;
         AG200_Sim : Bool;
         TT500_HH_Alarm : Bool;
         TT500_H_Alarm : Bool;
         TT500_L_Alarm : Bool;
         TT500_LL_Alarm : Bool;
         TT500_Chan_Fail : Bool;
         TT500_Sim : Bool;
      END_STRUCT;
      Commands : Struct
         PT100_Scal_Min_Eu : Real;   // PT100 Нижняя шкала в инж. единицах
         PT100_Scal_Max_Eu : Real;   // PT100 Верхняя шкала в инж. единицах
         PT100_HH_Lim : Real;   // PT100 ВАУ
         PT100_H_Lim : Real;   // PT100 ВПУ
         PT100_L_Lim : Real;   // PT100 НПУ
         PT100_LL_Lim : Real;   // PT100 НАУ
         PT100_Sim_Value : Real;   // PT100 Симуляционное значение
         TT100_Scal_Min_Eu : Real;   // TT100 Нижняя шкала в инж. единицах
         TT100_Scal_Max_Eu : Real;   // TT100 Верхняя шкала в инж. единицах
         TT100_HH_Lim : Real;   // TT100 ВАУ
         TT100_H_Lim : Real;   // TT100 ВПУ
         TT100_L_Lim : Real;   // TT100 НПУ
         TT100_LL_Lim : Real;   // TT100 НАУ
         TT100_Sim_Value : Real;   // TT100 Симуляционное значение
         LT100_Scal_Min_Eu : Real;   // LT100 Нижняя шкала в инж. единицах
         LT100_Scal_Max_Eu : Real;   // LT100 Верхняя шкала в инж. единицах
         LT100_HH_Lim : Real;   // LT100 ВАУ
         LT100_H_Lim : Real;   // LT100 ВПУ
         LT100_L_Lim : Real;   // LT100 НПУ
         LT100_LL_Lim : Real;   // LT100 НАУ
         LT100_Sim_Value : Real;   // LT100 Симуляционное значение
         AG100_Scal_Min_Eu : Real;   // AG100 Нижняя шкала в инж. единицах
         AG100_Scal_Max_Eu : Real;   // AG100 Верхняя шкала в инж. единицах
         AG100_HH_Lim : Real;   // AG100 ВАУ
         AG100_H_Lim : Real;   // AG100 ВПУ
         AG100_L_Lim : Real;   // AG100 НПУ
         AG100_LL_Lim : Real;   // AG100 НАУ
         AG100_Sim_Value : Real;   // AG100 Симуляционное значение
         PT200_Scal_Min_Eu : Real;   // PT200 Нижняя шкала в инж. единицах
         PT200_Scal_Max_Eu : Real;   // PT200 Верхняя шкала в инж. единицах
         PT200_HH_Lim : Real;   // PT200 ВАУ
         PT200_H_Lim : Real;   // PT200 ВПУ
         PT200_L_Lim : Real;   // PT200 НПУ
         PT200_LL_Lim : Real;   // PT200 НАУ
         PT200_Sim_Value : Real;   // PT200 Симуляционное значение
         TT200_Scal_Min_Eu : Real;   // TT200 Нижняя шкала в инж. единицах
         TT200_Scal_Max_Eu : Real;   // TT200 Верхняя шкала в инж. единицах
         TT200_HH_Lim : Real;   // TT200 ВАУ
         TT200_H_Lim : Real;   // TT200 ВПУ
         TT200_L_Lim : Real;   // TT200 НПУ
         TT200_LL_Lim : Real;   // TT200 НАУ
         TT200_Sim_Value : Real;   // TT200 Симуляционное значение
         LT200_Scal_Min_Eu : Real;   // LT200 Нижняя шкала в инж. единицах
         LT200_Scal_Max_Eu : Real;   // LT200 Верхняя шкала в инж. единицах
         LT200_HH_Lim : Real;   // LT200 ВАУ
         LT200_H_Lim : Real;   // LT200 ВПУ
         LT200_L_Lim : Real;   // LT200 НПУ
         LT200_LL_Lim : Real;   // LT200 НАУ
         LT200_Sim_Value : Real;   // LT200 Симуляционное значение
         AG200_Scal_Min_Eu : Real;   // AG200 Нижняя шкала в инж. единицах
         AG200_Scal_Max_Eu : Real;   // AG200 Верхняя шкала в инж. единицах
         AG200_HH_Lim : Real;   // AG200 ВАУ
         AG200_H_Lim : Real;   // AG200 ВПУ
         AG200_L_Lim : Real;   // AG200 НПУ
         AG200_LL_Lim : Real;   // AG200 НАУ
         AG200_Sim_Value : Real;   // AG200 Симуляционное значение
         TT500_Scal_Min_Eu : Real;   // TT500 Нижняя шкала в инж. единицах
         TT500_Scal_Max_Eu : Real;   // TT500 Верхняя шкала в инж. единицах
         TT500_HH_Lim : Real;   // TT500 ВАУ
         TT500_H_Lim : Real;   // TT500 ВПУ
         TT500_L_Lim : Real;   // TT500 НПУ
         TT500_LL_Lim : Real;   // TT500 НАУ
         TT500_Sim_Value : Real;   // TT500 Симуляционное значение
         PCV300_Setpoint : Real;   // PCV300 Уставка
         PCV300_ManualValue : Real;   // PCV300 Задание в ручном режиме
         PCV300_Gain : Real;   // PCV300 Коэфф. пропорциональности
         PCV300_Ti : Real;   // PCV300 Время интегрирования
         PCV300_Td : Real;   // PCV300 Время дифференциирования
         PCV300_TdFiltRatio : Real;   // PCV300 Зона нечувствительности
         PCV300_OutputUpperLimit : Real;   // PCV300 Верхнее ограничение хода
         PCV300_OutputLowerLimit : Real;   // PCV300 Нижнее ограничение хода
         LCV300_Setpoint : Real;   // LCV300 Уставка
         LCV300_ManualValue : Real;   // LCV300 Задание в ручном режиме
         LCV300_Gain : Real;   // LCV300 Коэфф. пропорциональности
         LCV300_Ti : Real;   // LCV300 Время интегрирования
         LCV300_Td : Real;   // LCV300 Время дифференциирования
         LCV300_TdFiltRatio : Real;   // LCV300 Зона нечувствительности
         LCV300_OutputUpperLimit : Real;   // LCV300 Верхнее ограничение хода
         LCV300_OutputLowerLimit : Real;   // LCV300 Нижнее ограничение хода
         PT100_HH_Alarm_En : Bool;   // PT100 Включить ВАУ
         PT100_H_Alarm_En : Bool;   // PT100 Включить ВПУ
         PT100_L_Alarm_En : Bool;   // PT100 Включить НПУ
         PT100_LL_Alarm_En : Bool;   // PT100 Включить НАУ
         PT100_Sim_En : Bool;   // PT100 Включить симуляцию
         TT100_HH_Alarm_En : Bool;   // TT100 Включить ВАУ
         TT100_H_Alarm_En : Bool;   // TT100 Включить ВПУ
         TT100_L_Alarm_En : Bool;   // TT100 Включить НПУ
         TT100_LL_Alarm_En : Bool;   // TT100 Включить НАУ
         TT100_Sim_En : Bool;   // TT100 Включить симуляцию
         LT100_HH_Alarm_En : Bool;   // LT100 Включить ВАУ
         LT100_H_Alarm_En : Bool;   // LT100 Включить ВПУ
         LT100_L_Alarm_En : Bool;   // LT100 Включить НПУ
         LT100_LL_Alarm_En : Bool;   // LT100 Включить НАУ
         LT100_Sim_En : Bool;   // LT100 Включить симуляцию
         AG100_HH_Alarm_En : Bool;   // AG100 Включить ВАУ
         AG100_H_Alarm_En : Bool;   // AG100 Включить ВПУ
         AG100_L_Alarm_En : Bool;   // AG100 Включить НПУ
         AG100_LL_Alarm_En : Bool;   // AG100 Включить НАУ
         AG100_Sim_En : Bool;   // AG100 Включить симуляцию
         PT200_HH_Alarm_En : Bool;   // PT200 Включить ВАУ
         PT200_H_Alarm_En : Bool;   // PT200 Включить ВПУ
         PT200_L_Alarm_En : Bool;   // PT200 Включить НПУ
         PT200_LL_Alarm_En : Bool;   // PT200 Включить НАУ
         PT200_Sim_En : Bool;   // PT200 Включить симуляцию
         TT200_HH_Alarm_En : Bool;   // TT200 Включить ВАУ
         TT200_H_Alarm_En : Bool;   // TT200 Включить ВПУ
         TT200_L_Alarm_En : Bool;   // TT200 Включить НПУ
         TT200_LL_Alarm_En : Bool;   // TT200 Включить НАУ
         TT200_Sim_En : Bool;   // TT200 Включить симуляцию
         LT200_HH_Alarm_En : Bool;   // LT200 Включить ВАУ
         LT200_H_Alarm_En : Bool;   // LT200 Включить ВПУ
         LT200_L_Alarm_En : Bool;   // LT200 Включить НПУ
         LT200_LL_Alarm_En : Bool;   // LT200 Включить НАУ
         LT200_Sim_En : Bool;   // LT200 Включить симуляцию
         AG200_HH_Alarm_En : Bool;   // AG200 Включить ВАУ
         AG200_H_Alarm_En : Bool;   // AG200 Включить ВПУ
         AG200_L_Alarm_En : Bool;   // AG200 Включить НПУ
         AG200_LL_Alarm_En : Bool;   // AG200 Включить НАУ
         AG200_Sim_En : Bool;   // AG200 Включить симуляцию
         TT500_HH_Alarm_En : Bool;   // TT500 Включить ВАУ
         TT500_H_Alarm_En : Bool;   // TT500 Включить ВПУ
         TT500_L_Alarm_En : Bool;   // TT500 Включить НПУ
         TT500_LL_Alarm_En : Bool;   // TT500 Включить НАУ
         TT500_Sim_En : Bool;   // TT500 Включить симуляцию
         PCV300_ManualEnable : Bool;   // PCV300 включить ручной режим
         LCV300_ManualEnable : Bool;   // LCV300 включить ручной режим
         GFU_Spark : Bool;   // Подать искру на ГФУ
         Head_cmd_on : Bool;   // Обогрев включить
         Head_cmd_off : Bool;   // Обогрев выключить
         Head_cmd_reset : Bool;   // Обогрев сброс ошибки
         Power_cmd_on : Bool;   // Питание установки включить
         Power_cmd_off : Bool;   // Питание установки выключить
         Power_cmd_reset : Bool;   // Питание установки сброс ошибки
         XV100_cmd_open : Bool;   // XV100 Команда открыть
         XV100_cmd_close : Bool;   // XV100 Команда закрыть
         XV100_cmd_reset : Bool;   // XV100 Команда сброс ошибки
      END_STRUCT;
   END_VAR
BEGIN
END_DATA_BLOCK

// folder: System blocks/Program resources

DATA_BLOCK "Timer_Busy_Modbus_Reg"   // DB17
{ S7_Optimized_Access := 'TRUE' }
AUTHOR : Simatic
FAMILY : IEC
NAME : IEC_TMR
VERSION : 1.0
// stored: InstanceOfName IEC_TIMER
"IEC_TIMER"
BEGIN
END_DATA_BLOCK

DATA_BLOCK "Timer_Busy_Modbus_Reg2"   // DB18
{ S7_Optimized_Access := 'TRUE' }
AUTHOR : Simatic
FAMILY : IEC
NAME : IEC_TMR
VERSION : 1.0
// stored: InstanceOfName IEC_TIMER
"IEC_TIMER"
BEGIN
END_DATA_BLOCK

DATA_BLOCK "Timer_Close_XV100"   // DB33
{ S7_Optimized_Access := 'TRUE' }
AUTHOR : Simatic
FAMILY : IEC
NAME : IEC_TMR
VERSION : 1.0
// stored: InstanceOfName IEC_TIMER
"IEC_TIMER"
BEGIN
END_DATA_BLOCK

DATA_BLOCK "Timer_Open_XV100"   // DB34
{ S7_Optimized_Access := 'TRUE' }
AUTHOR : Simatic
FAMILY : IEC
NAME : IEC_TMR
VERSION : 1.0
// stored: InstanceOfName IEC_TIMER
"IEC_TIMER"
BEGIN
END_DATA_BLOCK

DATA_BLOCK "UVP_off"   // DB35
{ S7_Optimized_Access := 'TRUE' }
AUTHOR : Simatic
FAMILY : IEC
NAME : IEC_TMR
VERSION : 1.0
// stored: InstanceOfName IEC_TIMER
"IEC_TIMER"
BEGIN
END_DATA_BLOCK

DATA_BLOCK "Spark_time"   // DB36
{ S7_Optimized_Access := 'TRUE' }
AUTHOR : Simatic
FAMILY : IEC
NAME : IEC_TMR
VERSION : 1.0
// stored: InstanceOfName IEC_TIMER
"IEC_TIMER"
BEGIN
END_DATA_BLOCK

// folder: (top level)

FUNCTION "In_Channel" : Void   // FC8, SCL
{ S7_Optimized_Access := 'TRUE' }
VERSION : 0.1
BEGIN
   // Обработка аналоговых сигналов
   "PT100"("AI1_Ch0");
   IF "PT100".Signal_AI.HH_Alarm THEN
       "PT100".Signal_AI.H_Alarm := false;
   END_IF;
   "TT100"("AI1_Ch1");
   "LT100"("AI1_Ch2");
   "AG100"("AI1_Ch3");
   "PT200"("AI1_Ch4");
   "TT200"("AI1_Ch5");
   "LT200"("AI1_Ch6");
   "AG200"("AI1_Ch7");
   "TT500"("AI2_Ch0");

   // Обработка дискретных входов
   "DI1"("DI1_In");
   "DI2"("DI2_In");
   "DI3"("DI3_In");
END_FUNCTION

FUNCTION "Out_Channel" : Void   // FC12, SCL
{ S7_Optimized_Access := 'TRUE' }
VERSION : 0.1
BEGIN
   // Выдача сигналов на дискретные выходы
   "DO1"("DO1_Out");
   "DO2"("DO2_Out");
END_FUNCTION

FUNCTION "Protect" : Void   // FC13, SCL
{ S7_Optimized_Access := 'TRUE' }
VERSION : 0.1
BEGIN
   // ***************************** Свето-звуковая сигнализация **************************************************************
   "DO1".Slot.Pins[0] := "AG100".Signal_AI.H_Alarm OR "AG200".Signal_AI.H_Alarm OR "DI2".Slot.Pins[5];
   "DO1".Slot.Pins[1] := "AG100".Signal_AI.HH_Alarm OR "AG200".Signal_AI.HH_Alarm;

   //если пришла аварийная загазованность и XV100 закрыта, вырубаем питание установки
   "Alarm_Gas" := "AG100".Signal_AI.HH_Alarm OR "AG200".Signal_AI.HH_Alarm;
   //IF ("Alarm_Gas" AND NOT "Alarm_Gas_prev") THEN
   IF ("Alarm_Gas" AND "DI3".Slot.Pins[5]) THEN
       "Power".Device.Cmd_Off := 4;
   END_IF;
   "Alarm_Gas_prev" := "Alarm_Gas"; // для определения фронта срабатывания загазованности

   // ***************************** ГФУ *********************************
   IF (NOT "CommandHMI_Spark_prev" AND "DATA".Commands.GFU_Spark) THEN
       "Spark_time".TON(IN := true, PT := t#10s);
   END_IF;
   IF ("Spark_time".Q AND "DATA".Commands.GFU_Spark) THEN
       "DATA".Commands.GFU_Spark := false;
       "Spark_time".TON (IN := false, PT := t#30s);
   END_IF;
   "CommandHMI_Spark_prev" := "DATA".Commands.GFU_Spark;

   "DO1".Slot.Pins[4] := "DI2".Slot.Pins[0] OR "DATA".Commands.GFU_Spark; // подача искры

   // ***************************** XV100 *********************************
   // Определение аварии для закрытия клапана - пересмотреть на ПНР, уточнить по РЭ
   //"Alarm_protect_XV100" := "PT100".Signal_AI.HH_Alarm OR "LT100".Signal_AI.HH_Alarm OR "AG100".Signal_AI.HH_Alarm OR "AG200".Signal_AI.HH_Alarm OR "DI1".Slot.Pins[0];
   "Alarm_protect_XV100" := "AG100".Signal_AI.HH_Alarm OR "AG200".Signal_AI.HH_Alarm;

   // закрываем клапан если есть авария или есть команда на закрытие или нажата кнопка аварийного останова и не закрыт
   IF NOT "DI3".Slot.Pins[5] AND ("Alarm_protect_XV100" OR "DATA".Commands.XV100_cmd_close OR "DI2".Slot.Pins[3]) THEN
       "DO1".Slot.Pins[3] := true;
   END_IF;
   "Alarm_protect_XV100_prev" := "Alarm_protect_XV100"; // для определения фронта срабатывания аварии

   // Определяем таймаут для исполнения команды закрытия
   "Timer_Close_XV100".TON(IN := "DO1".Slot.Pins[3], PT := t#30s);

   IF "Timer_Close_XV100".Q AND NOT "DI3".Slot.Pins[5] THEN
       "DATA".Measuring.XV100_no_cmd_close := true;
       "DO1".Slot.Pins[3] := false;
       "DATA".Commands.XV100_cmd_close := false;
       "Timer_Close_XV100".TON(IN := false, PT := t#30s);
   END_IF;

   // если есть сигнал на закрытие и пришел сигнал что Закрыто - снимаем команду
   IF "DO1".Slot.Pins[3] AND "DI3".Slot.Pins[5] THEN
       "DO1".Slot.Pins[3] := false;
       "DATA".Commands.XV100_cmd_close := false;
       "Timer_Close_XV100".TON(IN := false, PT := t#30s);
   END_IF;

   // открываем клапан если есть команда на открытие и не открыт и нет сигнала на закрытие и нет аварии и аварийного останова
   IF NOT "DI3".Slot.Pins[4] AND NOT "Alarm_protect_XV100" AND NOT "DI2".Slot.Pins[3] AND "DATA".Commands.XV100_cmd_open AND NOT "DO1".Slot.Pins[3] THEN
       "DO1".Slot.Pins[2] := true;
   END_IF;

   // Определяем таймаут для исполнения команды открытия
   "Timer_Open_XV100".TON(IN := "DO1".Slot.Pins[2], PT := t#30s);

   IF "Timer_Open_XV100".Q AND NOT "DI3".Slot.Pins[4] THEN
       "DATA".Measuring.XV100_no_cmd_open := true;
       "DO1".Slot.Pins[2] := false;
       "DATA".Commands.XV100_cmd_open := false;
       "Timer_Open_XV100".TON(IN := false, PT := t#30s);
   END_IF;

   // если есть сигнал на открытие и пришел сигнал что Открыто - снимаем команду
   IF "DO1".Slot.Pins[2] AND "DI3".Slot.Pins[4] THEN
       "DO1".Slot.Pins[2] := false;
       "DATA".Commands.XV100_cmd_open := false;
       "Timer_Open_XV100".TON(IN := false, PT := t#30s);
   END_IF;

   // Сброс ошибки
   IF "DATA".Commands.XV100_cmd_reset THEN
       "DATA".Measuring.XV100_no_cmd_close := false;
       "DATA".Measuring.XV100_no_cmd_open := false;
       "DO1".Slot.Pins[2] := false;
       "DO1".Slot.Pins[3] := false;
       "DATA".Commands.XV100_cmd_close := false;
       "DATA".Commands.XV100_cmd_open := false;
       "DATA".Commands.XV100_cmd_reset := false;
   END_IF;
END_FUNCTION

ORGANIZATION_BLOCK "Main"   // OB1, LAD, ProgramCycle
TITLE = "Main Program Sweep (Cycle)"
{ S7_Optimized_Access := 'TRUE' }
VERSION : 0.1
   VAR_INPUT
      Initial_Call : Bool;   // Initial call of this OB
      Remanence : Bool;   // =True, if remanent data are available
   END_VAR
BEGIN

REGION Network 1: Блок обработки входов
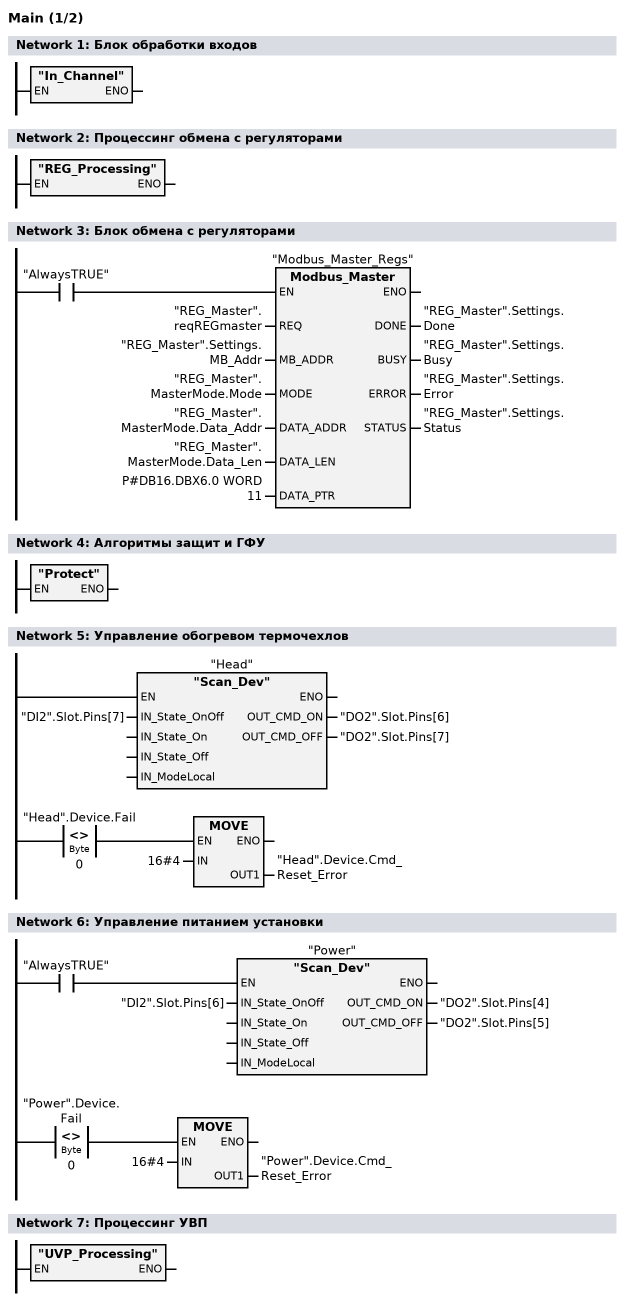
   RUNG wire#powerrail
      "In_Channel"()
   END_RUNG
   // the same network as SCL:
   "In_Channel"();
END_REGION

REGION Network 2: Процессинг обмена с регуляторами
   RUNG wire#powerrail
      "REG_Processing"()
   END_RUNG
   // the same network as SCL:
   "REG_Processing"();
END_REGION

REGION Network 3: Блок обмена с регуляторами
   IF "AlwaysTRUE" THEN
       "Modbus_Master_Regs"(REQ := "REG_Master".reqREGmaster,   // Modbus_Master
                            MB_ADDR := "REG_Master".Settings.MB_Addr,
                            MODE := "REG_Master".MasterMode.Mode,
                            DATA_ADDR := "REG_Master".MasterMode.Data_Addr,
                            DATA_LEN := "REG_Master".MasterMode.Data_Len,
                            DATA_PTR := P#DB16.DBX6.0 WORD 11,
                            DONE => "REG_Master".Settings.Done,
                            BUSY => "REG_Master".Settings.Busy,
                            ERROR => "REG_Master".Settings.Error,
                            STATUS => "REG_Master".Settings.Status);
   END_IF;
END_REGION

REGION Network 4: Алгоритмы защит и ГФУ
   RUNG wire#powerrail
      "Protect"()
   END_RUNG
   // the same network as SCL:
   "Protect"();
END_REGION

REGION Network 5: Управление обогревом термочехлов
   RUNG wire#powerrail
      "Head"(IN_State_OnOff := "DI2".Slot.Pins[7], IN_State_On :=, IN_State_Off :=, IN_ModeLocal :=, OUT_CMD_ON => "DO2".Slot.Pins[6], OUT_CMD_OFF => "DO2".Slot.Pins[7])
   END_RUNG
   RUNG wire#powerrail
      { S7_Templates := "SrcType := Byte" } NE_Contact(in1 := "Head".Device.Fail, in2 := 0)
      Move(in := 16#4, out1 => "Head".Device.Cmd_Reset_Error)
   END_RUNG
   // the same network as SCL:
   "Head"(IN_State_OnOff := "DI2".Slot.Pins[7],   // "Scan_Dev"
          OUT_CMD_ON => "DO2".Slot.Pins[6],
          OUT_CMD_OFF => "DO2".Slot.Pins[7]);
   IF "Head".Device.Fail <> 0 THEN "Head".Device.Cmd_Reset_Error := 16#4; END_IF;
END_REGION

REGION Network 6: Управление питанием установки
   RUNG wire#powerrail
      Contact( "AlwaysTRUE" )
      "Power"(IN_State_OnOff := "DI2".Slot.Pins[6], IN_State_On :=, IN_State_Off :=, IN_ModeLocal :=, OUT_CMD_ON => "DO2".Slot.Pins[4], OUT_CMD_OFF => "DO2".Slot.Pins[5])
   END_RUNG
   RUNG wire#powerrail
      { S7_Templates := "SrcType := Byte" } NE_Contact(in1 := "Power".Device.Fail, in2 := 0)
      Move(in := 16#4, out1 => "Power".Device.Cmd_Reset_Error)
   END_RUNG
   // the same network as SCL:
   IF "AlwaysTRUE" THEN
       "Power"(IN_State_OnOff := "DI2".Slot.Pins[6],   // "Scan_Dev"
               OUT_CMD_ON => "DO2".Slot.Pins[4],
               OUT_CMD_OFF => "DO2".Slot.Pins[5]);
   END_IF;
   IF "Power".Device.Fail <> 0 THEN "Power".Device.Cmd_Reset_Error := 16#4; END_IF;
END_REGION

REGION Network 7: Процессинг УВП
   RUNG wire#powerrail
      "UVP_Processing"()
   END_RUNG
   // the same network as SCL:
   "UVP_Processing"();
END_REGION

REGION Network 8: Блок обмена с УВП
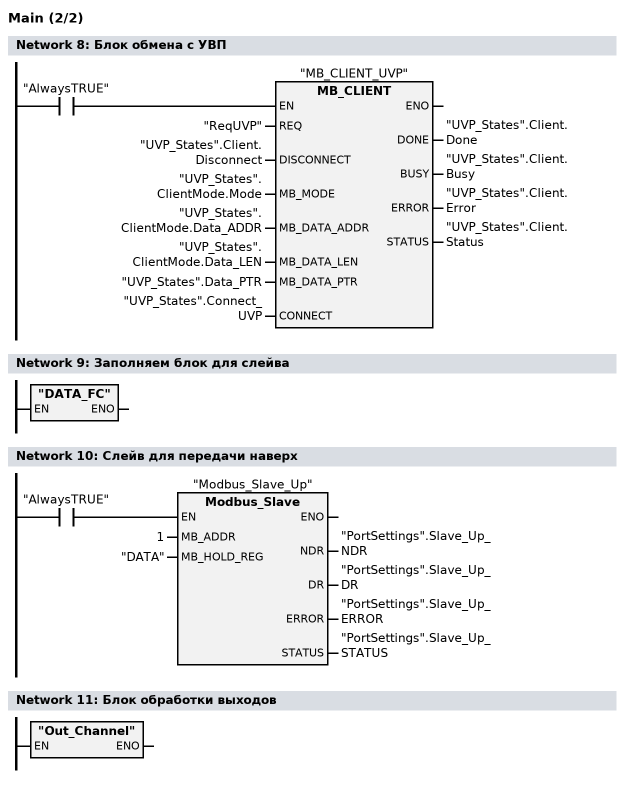
   IF "AlwaysTRUE" THEN
       "MB_CLIENT_UVP"(REQ := "ReqUVP",   // MB_CLIENT
                       DISCONNECT := "UVP_States".Client.Disconnect,
                       MB_MODE := "UVP_States".ClientMode.Mode,
                       MB_DATA_ADDR := "UVP_States".ClientMode.Data_ADDR,
                       MB_DATA_LEN := "UVP_States".ClientMode.Data_LEN,
                       MB_DATA_PTR := "UVP_States".Data_PTR,
                       CONNECT := "UVP_States".Connect_UVP,
                       DONE => "UVP_States".Client.Done,
                       BUSY => "UVP_States".Client.Busy,
                       ERROR => "UVP_States".Client.Error,
                       STATUS => "UVP_States".Client.Status);
   END_IF;
END_REGION

REGION Network 9: Заполняем блок для слейва
   RUNG wire#powerrail
      "DATA_FC"()
   END_RUNG
   // the same network as SCL:
   "DATA_FC"();
END_REGION

REGION Network 10: Слейв для передачи наверх
   IF "AlwaysTRUE" THEN
       "Modbus_Slave_Up"(MB_ADDR := 1,   // Modbus_Slave
                         MB_HOLD_REG := "DATA",
                         NDR => "PortSettings".Slave_Up_NDR,
                         DR => "PortSettings".Slave_Up_DR,
                         ERROR => "PortSettings".Slave_Up_ERROR,
                         STATUS => "PortSettings".Slave_Up_STATUS);
   END_IF;
END_REGION

REGION Network 11: Блок обработки выходов
   RUNG wire#powerrail
      "Out_Channel"()
   END_RUNG
   // the same network as SCL:
   "Out_Channel"();
END_REGION
END_ORGANIZATION_BLOCK

ORGANIZATION_BLOCK "Cyclic100msec"   // OB30, SCL, CyclicInterrupt
{ S7_Optimized_Access := 'TRUE' }
VERSION : 0.1
   VAR_INPUT
      Initial_Call : Bool;   // Initial call of this OB
      Event_Count : Int;   // Events discarded
   END_VAR
   VAR_TEMP
      real1 : Real;
      real2 : Real;
   END_VAR
BEGIN
   IF "PCV300".Reset = true THEN
       "PCV300".Reset := false;
   END_IF;
   // Безударный переход на ручной режим
   IF NOT "PCV300".ManualEnable THEN
       "PCV300".ManualValue := "PCV300".Output;
   END_IF;
   "PCV300"(
           //**************Значение процесса - поменять каждому регулятору**********************
            Input := "PT100".Signal_AI.Value,
           //**************Значение управляющего воздействия - поменять каждому регулятору**********************
           Output => #real1);



   IF "LCV300".Reset = true THEN
       "LCV300".Reset := false;
   END_IF;
   // Безударный переход на ручной режим
   IF NOT "LCV300".ManualEnable THEN
       "LCV300".ManualValue := "LCV300".Output;
   END_IF;
   "LCV300"(
           //**************Значение процесса - поменять каждому регулятору**********************
            Input := "LT100".Signal_AI.Value,
           //**************Значение управляющего воздействия - поменять каждому регулятору**********************
           Output => #real2);

   "REG_Data".PCV300_Setpoint := REAL_TO_INT(#real1) * 10;
   "REG_Data".LCV300_Setpoint := REAL_TO_INT(#real2) * 10;

   //
   "Regs".PCV300_Midle := "REG_Data".PCV300_Status.Intermediate_position;
   "Regs".PCV300_Alarm := "REG_Data".PCV300_Message.Error OR "REG_Data".PCV300_Status.Error;
   "Regs".PCV300_Warning := "REG_Data".PCV300_Message.Warning OR "REG_Data".PCV300_Status.Warning;
   "Regs".PCV300_Remont := false;
   "Regs".LCV300_Midle := "REG_Data".LCV300_Status.Intermediate_position;
   "Regs".LCV300_Alarm := "REG_Data".LCV300_Message.Error OR "REG_Data".LCV300_Status.Error;
   "Regs".LCV300_Warning := "REG_Data".LCV300_Message.Warning OR "REG_Data".LCV300_Status.Warning;
   "Regs".LCV300_Remont := false;

   IF "REG_Data".PCV300_Setpoint > 1000 THEN
       "REG_Data".PCV300_Setpoint := 1000;
   END_IF;
   IF "REG_Data".PCV300_Setpoint < 0 THEN
       "REG_Data".PCV300_Setpoint := 0;
   END_IF;

   IF "REG_Data".LCV300_Setpoint > 1000 THEN
       "REG_Data".LCV300_Setpoint := 1000;
   END_IF;
   IF "REG_Data".LCV300_Setpoint < 0 THEN
       "REG_Data".LCV300_Setpoint := 0;
   END_IF;


   // Запись в реманентные переменные уставок и параметров регуляторов
   "Regs".PCV300_Man_En := "PCV300".ManualEnable;
   "Regs".LCV300_Man_En := "LCV300".ManualEnable;

   "Regs".PCV300_Man_Value := "PCV300".ManualValue;
   "Regs".LCV300_Man_Value := "LCV300".ManualValue;

   "Regs".PCV300_SP := "PCV300".Setpoint;
   "Regs".LCV300_SP := "LCV300".Setpoint;

   "Regs".PCV300_OutputUpperLimit := "PCV300".Config.OutputUpperLimit;
   "Regs".LCV300_OutputUpperLimit := "LCV300".Config.OutputUpperLimit;

   "Regs".PCV300_OutputLowerLimit := "PCV300".Config.OutputLowerLimit;
   "Regs".LCV300_OutputLowerLimit := "LCV300".Config.OutputLowerLimit;
END_ORGANIZATION_BLOCK

ORGANIZATION_BLOCK "Startup"   // OB100, SCL, Startup
TITLE = "Complete Restart"
{ S7_Optimized_Access := 'TRUE' }
VERSION : 0.1
   VAR_INPUT
      LostRetentive : Bool;   // True if retentive data are lost
      LostRTC : Bool;   // True if date and time are lost
   END_VAR
BEGIN
   "Modbus_init"();  // Инициализация параметров Modbus

   // Чтение из реманентных переменных уставок и параметров регуляторов
   "PCV300".ManualEnable := "Regs".PCV300_Man_En;
   "LCV300".ManualEnable := "Regs".LCV300_Man_En;
   "PCV300".ManualValue := "Regs".PCV300_Man_Value;
   "LCV300".ManualValue := "Regs".LCV300_Man_Value;
   "PCV300".Setpoint := "Regs".PCV300_SP;
   "LCV300".Setpoint := "Regs".LCV300_SP;
   "PCV300".Config.OutputUpperLimit := "Regs".PCV300_OutputUpperLimit;
   "LCV300".Config.OutputUpperLimit := "Regs".LCV300_OutputUpperLimit;
   "PCV300".Config.OutputLowerLimit := "Regs".PCV300_OutputLowerLimit;
   "LCV300".Config.OutputLowerLimit := "Regs".LCV300_OutputLowerLimit;

   // Обогрев
   "Head".Device.Cfg_OutputLevelCmd := false;  // Тип управления: false-импульсное, true-постоянное
   "Head".Device.Cfg_TwoStateInputs := false;  // Число входов состояния устройства: True - 2 параметра, False - 1 параметр
   "Head".Device.Cfg_Time_OnOff := T#7s;
   "Head".Device.RunTime_LastScan := DT#1990-01-01-00:00:00;
   "Head".Cfg_Time_OnOff := 4;
   // Питание
   "Power".Device.Cfg_OutputLevelCmd := false;  // Тип управления: false-импульсное, true-постоянное
   "Power".Device.Cfg_TwoStateInputs := false;  // Число входов состояния устройства: True - 2 параметра, False - 1 параметр
   "Power".Device.Cfg_Time_OnOff := T#7s;
   "Power".Device.RunTime_LastScan := DT#1990-01-01-00:00:00;
   "Power".Cfg_Time_OnOff := 4;

   "DI1".Slot.Input_En := 16#FF;
   "DI2".Slot.Input_En := 16#FF;
   "DI2".Slot.Invert_En := 16#C0;
   "DI3".Slot.Input_En := 16#FF;


   "DO1".Slot.Output_En := 16#FFFF;
   "DO1".Slot.UsePinsAsInput := true;
   "DO2".Slot.Output_En := 16#FFFF;
   "DO2".Slot.UsePinsAsInput := true;
END_ORGANIZATION_BLOCK

// folder: FBs

FUNCTION_BLOCK "Scan_AI"   // FB1, SCL
TITLE = Analog input module block (current inputs)
{ S7_Optimized_Access := 'FALSE' }
NAME : Scan_AI
VERSION : 1.3
   VAR_INPUT
      CODE_ACP : Word := 0;   // Input ADC code
   END_VAR
   VAR
      Signal_AI : "dt_AI";
      HH_Timer : TON_TIME;
      H_Timer : TON_TIME;
      L_Timer : TON_TIME;
      LL_Timer : TON_TIME;
   END_VAR
   VAR_TEMP
      ACP_min : DInt;
      ACP_max : DInt;
      ACP_sc : DInt;   // Overload or shortcut code
      ACP_br : DInt;   // Negative overload or breakoff code
      Curr0_20_min : Real;
      Curr0_20_max : Real;
      Curr0_20_sc : Real;   // Overload or shortcut
      Curr0_20_br : Real;   // Negative overload or breakoff
      Curr4_20_min : Real;
      Curr4_20_max : Real;
      Curr4_20_sc : Real;   // Overload or shortcut
      Curr4_20_br : Real;   // Negative overload or breakoff TEMP
      Volt0_10_min : Real;
      Volt0_10_max : Real;
      Volt0_10_sc : Real;
      Temp_Real : Real;
      Temp_Int : Int;
      Temp_Start_Timer : Bool;
      Temp_Timer_State : Bool;
      temp_Min_Eu : Real;
      UEL : Byte;   // ВАУ
      UWL : Byte;   // ВПУ
      DWL : Byte;   // НПУ
      DEL : Byte;   // НАУ
      PNC : Byte;   // Параметр не контроллируется
      SIM : Byte;   // Симуляция
      MSK : Byte;   // Маскирование
      TST : Byte;   // Тестирование
   END_VAR
BEGIN

   // CONST
   //   ADC codes for Simatic S300
   //   Êîä ÀÖÏ     0-20  ìÀ    4-20  ìÀ     0-10 Â        Comment
   //    32512   |  23.52 ìÀ  | 22.81 ìÀ  |  11.759 Â  | Overload or shortcut
   //    27648   |  20.0  ìÀ  | 20.0  ìÀ  |  10.0 Â    | Normal
   //      1     |  723.4 íÀ  | 4.578 ìÀ  |  361.7 ìêÂ | Normal
   //      0     |    0.0 ìÀ  |   4   ìÀ  |  0.0 Â     | Normal
   //    -4865   |  -3.52 ìÀ  | 1.185 ìÀ  |  ----      | Negative overload or breakoff 
   #ACP_min := 0;
   #ACP_max := 27648;
   #ACP_sc := 32512;  // Overload or shortcut code
   #ACP_br := -4865;  // Negative overload or breakoff code (circuit only)
   #Curr0_20_min := 0.0;
   #Curr0_20_max := 20.0;
   #Curr0_20_sc := 23.52;  // Overload or shortcut
   #Curr0_20_br := -3.52;  // Negative overload or breakoff
   #Curr4_20_min := 4.0;
   #Curr4_20_max := 20.0;
   #Curr4_20_sc := 22.81;  // Overload or shortcut
   #Curr4_20_br := 1.185;  // Negative overload or breakoff
   #Volt0_10_min := 0.0;
   #Volt0_10_max := 10.0;
   #Volt0_10_sc := 11.759;

   #UEL := 2#00000001;
   #UWL := 2#00000010;
   #DWL := 2#00000100;
   #DEL := 2#00001000;
   #PNC := 2#00010000;
   #SIM := 2#00100000;
   #MSK := 2#01000000;
   #TST := 2#10000000;

   // 1) Îáÿçàòåëüíî ïîäàòü íà âõîä CODE_ACP çíà÷åíèå ñ ñîîòâåòñòâóþùåãî êàíàëà àíàëîãîâîãî ââîäà
   // 2) Îáÿçàòåëüíî âûñòàâèòü òèï ìàñøòàáèðîâàíèÿ Scale_Type, 1 ýòî 0-20 ìÀ à 0 ýòî 4-20 ìÀ 
   // 3) Îáÿçàòåëüíî âûñòàâèòü äèàïàçîíû ìàñøòàáèðîâàíèÿ Scal_Max_Eu è Scal_Min_Eu
   // 4) Âûñòàâèòü åñëè íåîáõîäèìî êîýôôèöèåíò ôèëüòðàöèè  K_filtr
   // 5) Ïðîâåðèòü ÷òî íå âêëþ÷åí ðåæèì ñèìóëÿöèè  Sim_En 


   //*   Ôîðìóëû ìàñøòàáèðîâàíèÿ:
   //*   Y = (X – Xmin ) * ( Ymax - Ymin ) / ( Xmax - Xmin ) + Ymin
   //*   X = (Y – Ymin ) * ( Xmax - Xmin ) / ( Ymax - Ymin ) + Xmin

   //------------------------------------------------------------------------
   //------------------Áëîê ðåæèìà ñèìóëÿöèè---------------------------------
   //------------------------------------------------------------------------ 

   //Åñëè ðåæèì ñèìóëÿöèè âêëþ÷åí òî èñïîëüçóåì çíà÷åíèå Sim_Value
   IF #Signal_AI.Sim_En THEN
       // Ìàñøòàáèðóåì çíà÷åíèå ñèìóëÿöèè â êîä ÀÖÏ - íå èñïîëüçóåòñÿ, òàê êàê èç-çà ðàçíûõ ðåæèìîâ 
       //  (òîê 4-20/0-20, íàïðÿæåíèå) ñëîæíî îäíîçíà÷íî ñäåëàòü ïðåîáðàçîâàíèå â ñîîòâåòñòâóþùóþ âåëèöèíó ÀÖÏ
       //#Signal_AI.Acp := ROUND (( #Signal_AI.Sim_Value - #Signal_AI.Scal_Min_Eu)*DINT_TO_REAL(#ACP_max - #ACP_min) /
       //                         ( #Signal_AI.Scal_Max_Eu - #Signal_AI.Scal_Min_Eu) + DINT_TO_REAL(#ACP_min));
       #Signal_AI.State := #Signal_AI.State OR #SIM;
       #Temp_Real := #Signal_AI.Sim_Value;
   ELSE
       // èíà÷å èñïîëüçóåì àíàëîãîâûé âõîä
       #Signal_AI.State := #Signal_AI.State AND (NOT (#SIM));
       #Signal_AI.Acp := WORD_TO_INT(#CODE_ACP);

       //------------------------------------------------------------------------
       //-------------Áëîê ìàñøòàáèðîâàíèÿ---------------------------------------
       //------------------------------------------------------------------------
       IF #Signal_AI.VoltageInputType THEN
           // âõîä íàïðÿæåíèÿ
           // îïðåäåëåíèå íàïðÿæåíèÿ èç êîäà àöï  
           #Signal_AI.Voltage := DINT_TO_REAL(#Signal_AI.Acp - #ACP_min) * (#Volt0_10_max - #Volt0_10_min) / (DINT_TO_REAL(#ACP_max - #ACP_min)) + #Volt0_10_min;
           // îïðåäåëèì ýêâèâàëåíò òîêà ÷åðåç âõîäíîå ñîïðîòèâëåíèå
           IF #Signal_AI.Resistance > 0 THEN
               #Signal_AI.Circuit := #Signal_AI.Voltage / #Signal_AI.Resistance;
               // îïðåäåëåíèå çíà÷åíèÿ ñèãíàëà â èíæ. âåëè÷èíå èç ýêâèâàëåíòà òîêà 
               IF #Signal_AI.Scale_0_20mA THEN
                   #Temp_Real := (#Signal_AI.Circuit - #Curr0_20_min) * (#Signal_AI.Scal_Max_Eu - #Signal_AI.Scal_Min_Eu) / (#Curr0_20_max - #Curr0_20_min) + #Signal_AI.Scal_Min_Eu;
               ELSE
                   #Temp_Real := (#Signal_AI.Circuit - #Curr4_20_min) * (#Signal_AI.Scal_Max_Eu - #Signal_AI.Scal_Min_Eu) / (#Curr4_20_max - #Curr4_20_min) + #Signal_AI.Scal_Min_Eu;
               END_IF;
           ELSE
               // îïðåäåëåíèå çíà÷åíèÿ ñèãíàëà â èíæ. âåëè÷èíå èç êîäà àöï 
               #Temp_Real := DINT_TO_REAL(#Signal_AI.Acp - #ACP_min) * (#Signal_AI.Scal_Max_Eu - #Signal_AI.Scal_Min_Eu) / (DINT_TO_REAL(#ACP_max - #ACP_min)) + #Signal_AI.Scal_Min_Eu;
           END_IF;

       ELSE
           // òîêîâûé âõîä
           IF #Signal_AI.Scale_0_20mA THEN          // Åñëè òèï ìàñøòàáèðîâàíèÿ 0-20 ìÀ òî
               // îïðåäåëåíèå òîêà èç êîäà àöï 
               #Signal_AI.Circuit := DINT_TO_REAL(#Signal_AI.Acp - #ACP_min) * (#Curr0_20_max - #Curr0_20_min) / (DINT_TO_REAL(#ACP_max - #ACP_min)) + #Curr0_20_min;
           ELSE                                    // Èíà÷å åñëè òèï ìàñøòàáèðîâàíèÿ 4-20 ìÀ òî
               // îïðåäåëåíèå òîêà èç êîäà àöï  
               #Signal_AI.Circuit := DINT_TO_REAL(#Signal_AI.Acp - #ACP_min) * (#Curr4_20_max - #Curr4_20_min) / (DINT_TO_REAL(#ACP_max - #ACP_min)) + #Curr4_20_min;
           END_IF;

           // îïðåäåëåíèå çíà÷åíèÿ ñèãíàëà â èíæ. âåëè÷èíå èç êîäà àöï
           IF (#Signal_AI.Scale_0_20mA AND #Signal_AI.Input_4mA_on_0_20mA) THEN// Åñëè äàò÷èê 4-20ìÀ èñïîëüçóåòñÿ íà âõîäå 0-20ìÀ
               // ñäâèãàåì âíèç íà 25% íèæíèé ïðåäåë äàò÷èêà, äî 0ìÀ 
               #temp_Min_Eu := #Signal_AI.Scal_Min_Eu - ((#Signal_AI.Scal_Max_Eu - #Signal_AI.Scal_Min_Eu) / 4.0);
               #Temp_Real := DINT_TO_REAL(#Signal_AI.Acp - #ACP_min) * (#Signal_AI.Scal_Max_Eu - #temp_Min_Eu) / (DINT_TO_REAL(#ACP_max - #ACP_min)) + #temp_Min_Eu;
           ELSE
               #Temp_Real := DINT_TO_REAL(#Signal_AI.Acp - #ACP_min) * (#Signal_AI.Scal_Max_Eu - #Signal_AI.Scal_Min_Eu) / (DINT_TO_REAL(#ACP_max - #ACP_min)) + #Signal_AI.Scal_Min_Eu;
           END_IF;
       END_IF;


   END_IF;

   //------------------------------------------------------------------------
   //-----------Áëîê ôèëüòðàöèè (ñãëàæèâàíèÿ) àíàëîãîâîãî ñèãíàëà------------
   // Åñëè ðåæèì ôèëüòðàöèè âêëþ÷åí ðàñ÷èòàòü çíà÷åíèå ïî ôîðìóëå Óâûõ=Óïîñë + Êôèëòð*( Óòåê - Óïîñë)
   // ïðè ñãëàæèâàíèè ïî íèæåïðèâåäåííîé  ôîðìóëå ïðîèñõîäèò ïîñêàíîâîå ïðèáëèæåíèå âûõîäíîãî
   // çíà÷åíèÿ ê òåêóùåìó (ðåàëüíîìó) ñèãíàëó
   //------------------------------------------------------------------------

   IF #Signal_AI.K_filtr > 0 THEN
       #Signal_AI.Value := #Signal_AI.Value_LastScan + #Signal_AI.K_filtr * (#Temp_Real - #Signal_AI.Value_LastScan);
       //Çàïîìèíàåì òåêóùåå çíà÷åíèå êàê çíà÷åíèå ñ ïîñëåäíåãî ñêàíà
       #Signal_AI.Value_LastScan := #Signal_AI.Value;
   ELSE
       // âûñòàâëÿåì òåêóùåå çíà÷åíèå 
       #Signal_AI.Value := #Temp_Real;
   END_IF;

   //------------------------------------------------------------------------
   //Áëîê ïðîâåðêè âûõîäà çíà÷åíèÿ ñèãíàëà èç ðàáî÷åãî äèàïàçîíà-------------
   //------------------------------------------------------------------------

   IF #Signal_AI.Value > #Signal_AI.Scal_Max_Eu THEN      //Ïðè âûõîäå çíà÷åíèÿ ñèãíàëà èç çàäàííîãî äèàïàçîíà ïðèðàâíèâàåì åãî ê âåðõíåìó ïðåäåëó ýòîãî äèàïàçîíà
       #Signal_AI.Value := #Signal_AI.Scal_Max_Eu;
       #Signal_AI.Scal_Max_Upper := true;                 //çàæèãàåì ôëàã ïðåâûøåíèÿ çíà÷åíèÿ ñèãíàëà âåðõíåãî ïðåäåëà äèàïàçîíà ìàñøòàáèðîâàíèÿ
   ELSE
       #Signal_AI.Scal_Max_Upper := false;
   END_IF;

   IF #Signal_AI.Value < #Signal_AI.Scal_Min_Eu THEN      //Ïðè âûõîäå çíà÷åíèÿ ñèãíàëà èç çàäàííîãî äèàïàçîíà ïðèðàâíèâàåì åãî ê íèæíåìó ïðåäåëó  ýòîãî äèàïàçîíà
       #Signal_AI.Value := #Signal_AI.Scal_Min_Eu;
       #Signal_AI.Scal_Min_Under := true;                 //çàæèãàåì ôëàã  çíà÷åíèÿ ñèãíàëà íèæå íèæíåãî ïðåäåëà äèàïàçîíà ìàñøòàáèðîâàíèÿ
   ELSE
       #Signal_AI.Scal_Min_Under := false;
   END_IF;

   //------------------------------------------------------------------------
   //---------Áëîê ïðîâåðêè ïðåâûøåíèÿ óñòàâêè ïî âåðõíåìó àâàðèéíîìó ïðåäåëó
   //------------------------------------------------------------------------
   IF #Signal_AI.HH_Alarm THEN    // Åñëè åñòü àâàðèÿ òî äëÿ îáåñïå÷åíèÿ ãèñòåðåçèñà 
       // Ðàçðåøåíèå íà ñòàðò òàéìåðà åñëè ïðîâåðêà ðàçðåøåíà è çíà÷åíèå ïðåâûøàåò óñòàâêó
       #Temp_Start_Timer := #Signal_AI.HH_Alarm_En AND (#Signal_AI.Value > (#Signal_AI.HH_Lim - #Signal_AI.HH_DeadBand));
   ELSE
       // Ðàçðåøåíèå íà ñòàðò òàéìåðà åñëè ïðîâåðêà ðàçðåøåíà è çíà÷åíèå ïðåâûøàåò óñòàâêó
       #Temp_Start_Timer := #Signal_AI.HH_Alarm_En AND (#Signal_AI.Value > (#Signal_AI.HH_Lim + #Signal_AI.HH_DeadBand));
   END_IF;

   #HH_Timer(IN := #Temp_Start_Timer // IN: BOOL
             ,
             PT := #Signal_AI.HH_Delay // IN: TIME
   );

   //åñëè  âðåìÿ çàäåðæêè èñòåêëî òî çàæèãàåì ôëàã àâàðèè , èíà÷å ãàñèì åãî
   IF #HH_Timer.Q THEN
       #Signal_AI.HH_Alarm := true;
       #Signal_AI.State := #Signal_AI.State OR #UEL;
   ELSE
       #Signal_AI.HH_Alarm := false;
       #Signal_AI.State := #Signal_AI.State AND (NOT (#UEL));
   END_IF;

   //------------------------------------------------------------------------
   //Áëîê ïðîâåðêè ïðåâûøåíèÿ óñòàâêè ïî âåðõíåìó ïðåäóïðåäèòåëüíîìó ïðåäåëó
   //------------------------------------------------------------------------
   IF #Signal_AI.H_Alarm THEN    // Åñëè åñòü àâàðèÿ òî äëÿ îáåñïå÷åíèÿ ãèñòåðåçèñà 
       // Ðàçðåøåíèå íà ñòàðò òàéìåðà åñëè ïðîâåðêà ðàçðåøåíà è çíà÷åíèå ïðåâûøàåò óñòàâêó
       #Temp_Start_Timer := #Signal_AI.H_Alarm_En AND (#Signal_AI.Value > (#Signal_AI.H_Lim - #Signal_AI.H_DeadBand));
   ELSE
       // Ðàçðåøåíèå íà ñòàðò òàéìåðà åñëè ïðîâåðêà ðàçðåøåíà è çíà÷åíèå ïðåâûøàåò óñòàâêó
       #Temp_Start_Timer := #Signal_AI.H_Alarm_En AND (#Signal_AI.Value > (#Signal_AI.H_Lim + #Signal_AI.H_DeadBand));
   END_IF;

   #H_Timer(IN := #Temp_Start_Timer // IN: BOOL
            ,
            PT := #Signal_AI.H_Delay // IN: TIME
   );

   //åñëè  âðåìÿ çàäåðæêè èñòåêëî òî çàæèãàåì ôëàã àâàðèè , èíà÷å ãàñèì åãî
   IF #H_Timer.Q THEN
       #Signal_AI.H_Alarm := true;
       #Signal_AI.State := #Signal_AI.State OR #UWL;
   ELSE
       #Signal_AI.H_Alarm := false;
       #Signal_AI.State := #Signal_AI.State AND (NOT (#UWL));
   END_IF;

   //------------------------------------------------------------------------
   //--Áëîê ïðîâåðêè ïðåâûøåíèÿ óñòàâêè ïî íèæíåìó ïðåäóïðåäèòåëüíîìó ïðåäåëó
   //------------------------------------------------------------------------
   IF #Signal_AI.L_Alarm THEN    // Åñëè åñòü àâàðèÿ òî äëÿ îáåñïå÷åíèÿ ãèñòåðåçèñà 
       #Temp_Start_Timer := #Signal_AI.L_Alarm_En AND (#Signal_AI.Value < (#Signal_AI.L_Lim + #Signal_AI.L_DeadBand));   // Ðàçðåøåíèå íà ñòàðò òàéìåðà åñëè ïðîâåðêà ðàçðåøåíà è çíà÷åíèå ïðåâûøàåò óñòàâêó
   ELSE
       #Temp_Start_Timer := #Signal_AI.L_Alarm_En AND (#Signal_AI.Value < (#Signal_AI.L_Lim - #Signal_AI.L_DeadBand));   // Ðàçðåøåíèå íà ñòàðò òàéìåðà åñëè ïðîâåðêà ðàçðåøåíà è çíà÷åíèå ïðåâûøàåò óñòàâêó
   END_IF;

   #L_Timer(IN := #Temp_Start_Timer // IN: BOOL
            ,
            PT := #Signal_AI.L_Delay // IN: TIME
   );

   //åñëè  âðåìÿ çàäåðæêè èñòåêëî òî çàæèãàåì ôëàã àâàðèè , èíà÷å ãàñèì åãî
   IF #L_Timer.Q THEN
       #Signal_AI.L_Alarm := true;
       #Signal_AI.State := #Signal_AI.State OR #DWL;
   ELSE
       #Signal_AI.L_Alarm := false;
       #Signal_AI.State := #Signal_AI.State AND (NOT (#DWL));
   END_IF;

   //------------------------------------------------------------------------
   //-------Áëîê ïðîâåðêè ïðåâûøåíèÿ óñòàâêè ïî íèæíåìó àâàðèéíîìó ïðåäåëó---
   //------------------------------------------------------------------------
   IF #Signal_AI.LL_Alarm THEN    // Åñëè åñòü àâàðèÿ òî äëÿ îáåñïå÷åíèÿ ãèñòåðåçèñà 
       #Temp_Start_Timer := #Signal_AI.LL_Alarm_En AND (#Signal_AI.Value < (#Signal_AI.LL_Lim + #Signal_AI.LL_DeadBand));   // Ðàçðåøåíèå íà ñòàðò òàéìåðà åñëè ïðîâåðêà ðàçðåøåíà è çíà÷åíèå ïðåâûøàåò óñòàâêó
   ELSE
       #Temp_Start_Timer := #Signal_AI.LL_Alarm_En AND (#Signal_AI.Value < (#Signal_AI.LL_Lim - #Signal_AI.LL_DeadBand));   // Ðàçðåøåíèå íà ñòàðò òàéìåðà åñëè ïðîâåðêà ðàçðåøåíà è çíà÷åíèå ïðåâûøàåò óñòàâêó
   END_IF;

   #LL_Timer(IN := #Temp_Start_Timer // IN: BOOL
             ,
             PT := #Signal_AI.LL_Delay // IN: TIME
   );

   //åñëè  âðåìÿ çàäåðæêè èñòåêëî òî çàæèãàåì ôëàã àâàðèè , èíà÷å ãàñèì åãî
   IF #LL_Timer.Q THEN
       #Signal_AI.LL_Alarm := true;
       #Signal_AI.State := #Signal_AI.State OR #DEL;
   ELSE
       #Signal_AI.LL_Alarm := false;
       #Signal_AI.State := #Signal_AI.State AND (NOT (#DEL));
   END_IF;

   //Определяем состояние маскирования
   IF (#Signal_AI.HH_Alarm_En AND #Signal_AI.H_Alarm_En AND #Signal_AI.L_Alarm_En AND #Signal_AI.LL_Alarm_En) THEN
       #Signal_AI.State := #Signal_AI.State AND (NOT (#MSK));// OR #MSK;
   ELSE
       #Signal_AI.State := #Signal_AI.State OR #MSK;// AND (NOT (#MSK));
   END_IF;


   //------------------------------------------------------------------------
   //------Áëîê ïðîâåðêè íà êîðîòêîå çàìûêàíèå è îáðûâ-----------------------
   //------------------------------------------------------------------------
   IF (NOT #Signal_AI.Sim_En) THEN
       // Ïðîâåðêà íà êîðîòêîå çàìûêàíèå.
       #Signal_AI.Short_Circuit := (#Signal_AI.Acp >= #ACP_sc);

       // Ïðîâåðêà íà îáðûâ.
       IF #Signal_AI.VoltageInputType AND (#Signal_AI.Resistance > 0) THEN
           // âõîä íàïðÿæåíèÿ ñ ïðåîáðàçîâàíèåì â òîêîâûé
           IF #Signal_AI.Scale_0_20mA THEN
               #Signal_AI.Break := (#Signal_AI.Circuit <= #Curr0_20_br);
           ELSE
               #Signal_AI.Break := (#Signal_AI.Circuit <= #Curr4_20_br);
           END_IF;
       ELSE
           // òîêîâûé âõîä
           IF (#Signal_AI.Scale_0_20mA AND #Signal_AI.Input_4mA_on_0_20mA) THEN
               #Signal_AI.Break := (#Signal_AI.Circuit <= #Curr4_20_br);
           ELSE
               #Signal_AI.Break := (#Signal_AI.Acp <= #ACP_br);
           END_IF;
       END_IF;


       //  Ïðè îáðûâå èëè êîðîòêîì çàìûêàíèè  ãàñèì ôëàãè ñðàáàòûâàíèÿ óñòàâîê
       IF (#Signal_AI.Short_Circuit OR #Signal_AI.Break) THEN
           #Signal_AI.HH_Alarm := false;
           #Signal_AI.H_Alarm := false;
           #Signal_AI.L_Alarm := false;
           #Signal_AI.LL_Alarm := false;
           #Signal_AI.Chan_Fail := true;
           #Signal_AI.State := #Signal_AI.State OR #PNC;
       ELSE
           #Signal_AI.Chan_Fail := false;
           #Signal_AI.State := #Signal_AI.State AND (NOT (#PNC));
       END_IF;

   ELSE
       #Signal_AI.Short_Circuit := false;
       #Signal_AI.Break := false;
       #Signal_AI.Chan_Fail := false;
   END_IF;

   // Режим маскирования (или тестирования ?) - ХЗ. сделал как-будто это одно и то же
   IF (#Signal_AI.Mask_mode) THEN
       #Signal_AI.HH_Alarm_Logic := false;
       #Signal_AI.H_Alarm_Logic := false;
       #Signal_AI.L_Alarm_Logic := false;
       #Signal_AI.LL_Alarm_Logic := false;
       #Signal_AI.Chan_Fail_Logic := false;
       #Signal_AI.Test_mode := true;
   ELSE
       #Signal_AI.HH_Alarm_Logic := #Signal_AI.HH_Alarm;
       #Signal_AI.H_Alarm_Logic := #Signal_AI.H_Alarm;
       #Signal_AI.L_Alarm_Logic := #Signal_AI.L_Alarm;
       #Signal_AI.LL_Alarm_Logic := #Signal_AI.LL_Alarm;
       #Signal_AI.Chan_Fail_Logic := #Signal_AI.Chan_Fail;
       #Signal_AI.Test_mode := false;
   END_IF;

   // Квитирование аварий по аналоговым параметрам (моргание на HMI)
   IF ((#Signal_AI.HH_Alarm AND NOT #Signal_AI.Ack_HH) OR (#Signal_AI.LL_Alarm AND NOT #Signal_AI.Ack_LL)) THEN
       #Signal_AI.Ack_Alarm := 1;
   ELSIF ((#Signal_AI.HH_Alarm AND #Signal_AI.Ack_HH) OR (#Signal_AI.LL_Alarm AND #Signal_AI.Ack_LL)) THEN
       #Signal_AI.Ack_Alarm := 2;
   ELSIF (NOT #Signal_AI.HH_Alarm AND NOT #Signal_AI.LL_Alarm) THEN
       #Signal_AI.Ack_Alarm := 0;
       #Signal_AI.Ack_HH := false;
       #Signal_AI.Ack_LL := false;
   END_IF;

   IF ((#Signal_AI.H_Alarm AND NOT #Signal_AI.Ack_H) OR (#Signal_AI.L_Alarm AND NOT #Signal_AI.Ack_L)) THEN
       #Signal_AI.Ack_Warning := 1;
   ELSIF ((#Signal_AI.H_Alarm AND #Signal_AI.Ack_H) OR (#Signal_AI.L_Alarm AND #Signal_AI.Ack_L)) THEN
       #Signal_AI.Ack_Warning := 2;
   ELSIF (NOT #Signal_AI.H_Alarm AND NOT #Signal_AI.L_Alarm) THEN
       #Signal_AI.Ack_Warning := 0;
       #Signal_AI.Ack_H := false;
       #Signal_AI.Ack_L := false;
   END_IF;

   // Закраска прямоугольников на HMI
   IF (#Signal_AI.Mask_mode) THEN
       #Signal_AI.State_color := 3;
   ELSIF (#Signal_AI.Chan_Fail) THEN
       #Signal_AI.State_color := 4;
   ELSIF (#Signal_AI.HH_Alarm OR #Signal_AI.LL_Alarm) THEN
       #Signal_AI.State_color := 2;
   ELSIF (#Signal_AI.H_Alarm OR #Signal_AI.L_Alarm) THEN
       #Signal_AI.State_color := 1;
   ELSE
       #Signal_AI.State_color := 0;
   END_IF;
END_FUNCTION_BLOCK

FUNCTION_BLOCK "Scan_Dev"   // FB2, SCL
{ S7_Optimized_Access := 'FALSE' }
NAME : Scan_Dev
VERSION : 1.2
   VAR_INPUT
      IN_State_OnOff : Bool;   // On/Off state of device (Common state input)
      IN_State_On : Bool;   // On state of device (Separate state inputs)
      IN_State_Off : Bool;   // Off state of device (Separate state inputs)
      IN_ModeLocal : Bool;   // 0 - local control, 1 - remote control (device switch)
   END_VAR
   VAR_OUTPUT
      OUT_CMD_ON : Bool;   // Switch On command
      OUT_CMD_OFF : Bool;   // Switch Off command
   END_VAR
   VAR
      Device : Struct
         Cmd_On : Byte;   // Switch On commands : 0-None, 1-local, 2-remote auto, 4-remote manual(SCADA), 8-remote manual(OP)
         Cmd_Off : Byte;   // Switch Off commands: 0-None, 1-local, 2-remote auto, 4-remote manual(SCADA), 8-remote manual(OP)
         Mode : Byte := 4;   // Operate mode: 1-local, 2-remote auto, 4-remote manual(SCADA), 8-remote manual(OP), 16-Repair
         Fail : Byte;   // Fail (0-None, 128-common failure)
         State : Byte;   // Device state (0-off,1-on, 128-undefine)
         Control_Lock : Byte;   // Outer protection lock of device (0 - no protection, can work)
         Cfg_Time_OnOff : Time := T#5S;   // switch time (second)
         Cfg_OutPulseLen : Time := T#3S;   // Command pulse delay (second)
         RunTime : Real := 0.0;   // Worktime from last start (second)
         RunTime_Total : Real := 0.0;   // Total Worktime from last reset (second)
         RunTime_LastScan : Date_And_Time;   // Intermediate worktime (DTL)
         Sim_State : Byte;   // Device simulating state (0-off,1-on, 128-undefine)
         Sim_En : Bool;   // Simulate enable
         On_Flag : Bool := FALSE;   // On command accepted
         Off_Flag : Bool := FALSE;   // Off command accapted
         On_output : Bool := 0;   // On output state
         Off_output : Bool := 0;   // Off output state
         Cfg_OutputLevelCmd : Bool := FALSE;   // Output command type: false-pulse, true-level
         Cfg_TwoStateInputs : Bool := FALSE;   // Number of device state inputs: false-one common input, true-two separate inputs
         Cfg_CalculateRuntime : Bool := TRUE;   // true - calculate worktime
         Cfg_IgnoreStateInputs : Bool := FALSE;   // true - execute commands in any device state
         Cmd_Reset_Error : Byte;
         Reset_Error_Flag : Bool;
         Reset_Error_Output : Bool;
         auto : Bool;
      END_STRUCT;
      Device_Timer : TON_TIME;
      Cfg_Time_OnOff : DInt;
      Cfg_Time_OnOff_1 : DInt;
   END_VAR
   VAR_TEMP
      Temp_Start_Timer : Bool;
      Temp_Timer_Counting : Bool;
      Temp_Reset_Timer : Bool;
      Temp_Timer_State : Bool;
      Temp_Int : Int;
      Temp_CurTime : Time;
      Temp_Time : Time;
      temp_dint : DInt;
      CurrentTime : Date_And_Time;
      curr_TOD : Time_Of_Day;
      BDR_flag_ON : Bool;
      BDR_flag_OFF : Bool;
   END_VAR
BEGIN

   // 0)При инициализации (в OB100) необходимо сбрасывать Device.RunTime_LastScan в DTL#1970-1-1-0:0:0.0, иначе будет врать наработка 
   // 1)Каждому устройству необходимо выставить время включения-отключения  устройства (Cfg_Time_OnOf)
   // 2)Каждому устройству необходимо выставить тип управления (Cfg_TypeControl), 0-импульное, 1-постоянное 
   // 3)Каждому устройству необходимо выставить время длительности выходного импульса (Cfg_Time_Imp), если используется импульсный тип управления.                                                                     *//
   // 4)Каждому устройству выставить число входных сигналов состояния устройства Cfg_TwoStateInputs (True - 2 параметра, False - 1 параметр)


   // Обработки режима симуляции и определения состояния устройства

   //Если режим симуляции включен то заменяем ходные значение на значение для симуляции   
   IF #Device.Sim_En THEN
       #Device.State := #Device.Sim_State;
   ELSE
       // Если два входа состояния устройства
       IF #Device.Cfg_TwoStateInputs THEN
           IF #IN_State_Off THEN
               #Device.State := 2#00000000;                 // Состояние, Устройство выключено
           END_IF;
           IF #IN_State_On THEN
               #Device.State := 2#00000001;                 // Состояние, Устройство включено
           END_IF;
           IF NOT (#IN_State_Off XOR #IN_State_On) THEN       // Концевики оба =1 или =0 то
               #Device.State := 2#10000000;                 // Состояние, устройство неопределено
               #Device.Fail := #Device.Fail OR 2#00000100;   // Код аварии (4) - неопределенное значение концевиков
           END_IF;
       ELSE
           // Если один вход состояния устройства
           IF #IN_State_OnOff THEN
               #Device.State := 2#00000001;                 // Состояние, Устройство включено
           ELSE
               #Device.State := 2#00000000;                 // Состояние, Устройство выключено
           END_IF;
       END_IF;

       // Если состояние от переключателя - местн. режим то устанавливаем его иначе скидываем
       IF #IN_ModeLocal THEN
           #Device.Mode := #Device.Mode OR 2#00000001;
       ELSE
           #Device.Mode := #Device.Mode AND 2#11111110;
       END_IF;
   END_IF;



   // Обработка команд в соответствии с выбранным режимом управления и наличия аварии

   #Temp_Reset_Timer := false;

   // Если нет внешней аварии для блокировки управления устройством то можно включать устройство
   IF (#Device.Control_Lock = 0) THEN

       // Если есть команда на включение и она соответствует режиму управления
       IF (#Device.Mode AND #Device.Cmd_On) <> 0 THEN
           // Если состояние устройство не включено или мы игнорируем состояние устройства
           IF ((#Device.State AND 2#00000001) = 0) OR (#Device.Cfg_IgnoreStateInputs) THEN
               // Если флаг по команде управления на включение не зажжен, то обработаем команду однократно
               IF NOT #Device.On_Flag THEN

                   #Device.Fail := 0;                    // Сброс внутренней аварии

                   #Device.On_output := TRUE;          // Однократно по полож. фронту зажигаем внутреннюю команду на включение устройства
                   #Device.On_Flag := TRUE;          // Однократно по полож. фронту зажигаем флаг сигнализации что команда прошла

                   #Device.Off_Flag := FALSE;        // Однократно по полож. фронту сбрасываем флаг сигнализации что команда прошла
                   #Device.Off_output := FALSE;        // Однократно по полож. фронту сбрасываем внутреннюю команду на выключение

                   #Temp_Reset_Timer := TRUE;            // Однократно по полож. фронту команды сбрасываем таймер работы устройства  

               END_IF;
           END_IF;
       ELSE
           #Device.On_Flag := FALSE;                // Однократно по полож. фронту сбрасываем флаг сигнализации что команда прошла
       END_IF;

       // Если есть команда на выключение и она соответствует режиму управления
       IF (#Device.Mode AND #Device.Cmd_Off) <> 0 THEN
           // Если состояние устройство не выключено или мы игнорируем состояние устройства
           IF ((#Device.State AND 2#00000001) <> 0) OR (#Device.Cfg_IgnoreStateInputs) THEN
               // Если флаг по команде управления на выключение не зажжен, то обработаем команду однократно                     
               IF NOT #Device.Off_Flag THEN

                   #Device.Fail := 0;                    // Сброс внутренней аварии

                   #Device.On_output := false;         // Однократно по полож. фронту сбрасываем внутреннюю команду на включение устройства
                   #Device.On_Flag := FALSE;         // Однократно по полож. фронту сбрасываем флаг сигнализации что команда прошла

                   #Device.Off_Flag := TRUE;         // Однократно по полож. фронту зажигаем флаг сигнализации что команда прошла
                   #Device.Off_output := TRUE;         // Однократно по полож. фронту зажигаем внутреннюю команду на выключение

                   #Temp_Reset_Timer := TRUE;            // Однократно по полож. фронту команды сбрасываем таймер работы устройства

               END_IF;
           END_IF;
       ELSE
           #Device.Off_Flag := FALSE;                // Однократно по полож. фронту сбрасываем флаг сигнализации что команда прошла
       END_IF;

   END_IF;     //  IF ( Device.Control_Lock = 0) THEN


   IF (#Device.Mode AND #Device.Cmd_Reset_Error) <> 0 THEN
       // Если флаг по команде управления на сброс аварии не зажжен, то обработаем команду однократно                     
       IF NOT #Device.Reset_Error_Flag THEN

           #Device.Reset_Error_Output := TRUE;   // Однократно по полож. фронту зажигаем внутреннюю команду на сброс аварии устройства
           #Device.Reset_Error_Flag := TRUE;     // Однократно по полож. фронту зажигаем флаг сигнализации что команда прошла

           #Temp_Reset_Timer := TRUE;            // Однократно по полож. фронту команды сбрасываем таймер работы устройства
           #Device.Fail := 0;
           #Device.Off_Flag := false;
           #Device.On_Flag := false;
       END_IF;

   END_IF;
   #Device.Reset_Error_Flag := FALSE;    // Однократно по полож. фронту сбрасываем флаг сигнализации что команда прошла

   // команды не должны висеть - сбрасываем всё, что есть
   #Device.Cmd_On := 0;
   #Device.Cmd_Off := 0;
   #Device.Cmd_Reset_Error := 0;






   // Инициализация таймера


   // признак того, что таймер запущен, но ещё не досчитал до конца
   #Temp_Timer_Counting := (NOT #Device_Timer.Q) AND (#Device_Timer.ET > T#0ms);

   // Разрешение на старт таймера если есть команды на включение/выключение
   #Temp_Start_Timer := (NOT #Temp_Reset_Timer) AND (#Device.On_output OR #Device.Off_output);
   #Device_Timer(IN := #Temp_Start_Timer      // IN: BOOL
                 ,
                 PT := #Device.Cfg_Time_OnOff // IN: TIME
                 ,
                 ET => #Temp_CurTime);    // OUT: TIME

   // Снимаем флаг сброса таймера
   IF #Temp_Reset_Timer THEN
       #Temp_Reset_Timer := FALSE;
   END_IF;

   (*IF #Device.Fail = 2#10000001 AND #BDR_flag_ON THEN
     #OUT_CMD_OFF    := 0;
     #BDR_flag_ON  := false;
   END_IF;

   IF #Device.Fail = 2#10000011 AND #BDR_flag_OFF THEN
     #OUT_CMD_ON    := 0;
     #BDR_flag_OFF  := false;
    END_IF;*)
    //Формирование выходов при постоянном и импульсном типе управления

    // Если тип управления постоянный сигнал
    IF #Device.Cfg_OutputLevelCmd THEN
        #OUT_CMD_ON := #Device.On_output;
        #OUT_CMD_OFF := #Device.Off_output;
    ELSE
        // Если тип управления импульсный сигнал                                                          
        // Формируем импульс длительностью Cfg_OutPulseLen, но не дольше работы таймера
        IF ((#Temp_CurTime <= #Device.Cfg_OutPulseLen) AND #Temp_Timer_Counting) THEN
            #OUT_CMD_ON := #Device.On_output;
            #OUT_CMD_OFF := #Device.Off_output;
        ELSE
            #OUT_CMD_ON := 0;
            #OUT_CMD_OFF := 0;
        END_IF;


    END_IF;


    // Проверка отработки команд

    //если  время на отработку команды вышло и устройство не включилось или не выключилось то зажигаем аварию
    IF (#Device_Timer.Q) THEN
        // есть команда на включение
        IF #Device.On_output THEN
            IF ((#Device.State AND 2#00000001) = 0) THEN    // устройство не включилось
                #Device.Fail := #Device.Fail OR 2#00000001;   // Код аварии (1) - истекло время отработки команды

                //#Device.Cmd_Off := 16#04;//условие необходимое для вклчючение насоса бдр (modbus rtu)

            END_IF;
            #Device.On_output := 0;

        END_IF;
        // есть команда на выключение
        IF #Device.Off_output THEN
            IF (#Device.State AND 2#00000001) <> 0 THEN      // устройство не выключилось
                #Device.Fail := #Device.Fail OR 2#00000011;   // Код аварии (3) - истекло время отработки команды  

                // #Device.Cmd_On := 16#04;//условие необходимое для вклчючение насоса бдр (modbus rtu)
            END_IF;
            #Device.Off_output := 0;


        END_IF;
    END_IF;


    (*
    // Наработка устройства

    // Считываем текущее время контроллера
    #Temp_Int := RD_LOC_T(#CurrentTime);

    // считаем наработку только когда уже инициализвано предыдущее время
    IF (#Device.RunTime_LastScan > DTL#1970-1-1-0:0:0.0) THEN
        // если следует считать наработку и устройство включено
        IF (#Device.Cfg_CalculateRuntime AND ((#Device.State AND 2#00000001) = 1)) THEN
            #temp_dint := T_DIFF(IN1 := #CurrentTime, IN2 := #Device.RunTime_LastScan);
            #Device.RunTime := #Device.RunTime + DINT_TO_REAL(#temp_dint) * 0.001;
            #Device.RunTime_Total := #Device.RunTime_Total + DINT_TO_REAL(#temp_dint) * 0.001;
        ELSE
            #Device.RunTime := 0.0;         // Сбрасываем время наработки с последнего включения  
        END_IF;
    END_IF;

    #Device.RunTime_LastScan := #CurrentTime;

    //------------------------------------------------------------------------------------------//

    IF #Device.Fail <> 0 THEN             // Если есть какая нить авария то зажигаем общую аварию бит 8
        #Device.Fail := #Device.Fail OR 2#10000000;
    END_IF;

    #Cfg_Time_OnOff_1 := TIME_TO_DINT(#Device.Cfg_Time_OnOff);
    IF #Cfg_Time_OnOff_1 <> #Cfg_Time_OnOff * 1000 THEN
        #Device.Cfg_Time_OnOff := #Cfg_Time_OnOff * 1000;
    END_IF;
    *)
END_FUNCTION_BLOCK

FUNCTION_BLOCK "Scan_DI08"   // FB3, SCL
TITLE = '8-bit DI module scan'
{ S7_Optimized_Access := 'TRUE' }
NAME : ScanDI08
VERSION : 1.2
   VAR_INPUT
      In : Byte;
   END_VAR
   VAR
      Slot : Struct
         Input_En : Byte;   // enable input mask
         Filter_En : Byte;   // filter mask
         Invert_En : Byte;   // invert mask
         Sim_En : Byte;   // simulate enable mask
         Sim_Value : Byte;   // simulate value
         Input : Byte;   // In after inverting
         Value : Byte;   // Result after enable and filtering
         Value_Last_Scan : Byte;   // intermediate value
         Pins : Array[0..7] of Bool;   // hardware pins (accordance byte order)
      END_STRUCT;
   END_VAR
   VAR_TEMP
      Temp : Byte;
      Temp_In : Byte;
      i : Int;
   END_VAR
BEGIN



   #Temp_In := #In;
   #Slot.Input := #Temp_In XOR #Slot.Invert_En;         // Èíâåðòèðîâàíèå ñèãíàëîâ 
   #Temp_In := #Slot.Input AND #Slot.Input_En;      // Ïðîõîäÿò  òîëüêî ðàçðåøåííûå ñèíàëû     
   #Temp := #Slot.Value_Last_Scan XOR #Temp_In;   // Âûäåëåíèå áèòîâ èçìåíèâøèõñÿ çà ïåðèîä òàéìàóòà
   #Temp := #Temp AND #Slot.Filter_En;            // Ïðîâåðÿåì íàëè÷èå ðàçðåøåíèÿ íà ôèëüòðîâàíèå îò äðåáåçãà
   #Slot.Value := #Slot.Value AND #Temp;                // Ñîõðàíÿåì áèòû êîòîðûå íå äîëæíû èçìåíèòñÿ è îáíóëÿåì âñå îñòàëüíûå
   #Temp := NOT #Temp;                           // Èíâåðòèðóåì
   #Temp := #Temp AND #Temp_In;                  // Èçìåíèâøèåñÿ áèòû îáíóëÿåìè à íå èçìåíèâøèåñÿ ñ ïîñëåäíåãî ñêàíà áèòû çàïîìèíàåì 
   #Slot.Value := #Slot.Value OR #Temp;                 // Ôîðìèðóåì âûõîä 
   #Slot.Value_Last_Scan := #Temp_In;                   // Çàïîìèíàåì òåêóùåå çíà÷åíèå êàê çíà÷åíèå ïîñëåäíåãî ñêàíà

   // Ïðè âêëþ÷åííîé ñèìóëÿöèè çàìåíÿåì èñõîäíîå çíà÷åíèå íà Sim_Value
   #Slot.Value := (#Slot.Sim_En AND #Slot.Sim_Value) OR ((NOT #Slot.Sim_En) AND #Slot.Value);

   FOR #i := 0 TO 7 DO
       #Slot.Pins[#i] := "GetBitByte"(Data := #Slot.Value,
                                      pos := #i);
   END_FOR;
END_FUNCTION_BLOCK

FUNCTION_BLOCK "Put_DO08"   // FB4, SCL
TITLE = 'Puts 8-bit DO module data to Q-output'
{ S7_Optimized_Access := 'TRUE' }
NAME : PutDO08
VERSION : 1.0
   VAR_OUTPUT
      Out : Byte;
   END_VAR
   VAR
      Slot : "dt_DO";
   END_VAR
   VAR_TEMP
      Temp : Byte;
      i : Int;
   END_VAR
BEGIN


   IF #Slot.UsePinsAsInput THEN
       FOR #i := 0 TO 7 DO
           "SetBitByte"(pos := #i,
                        value := #Slot.Pins[#i],
                        Data := #Slot.Data_to_out);
       END_FOR;
   END_IF;

   #Temp := #Slot.Data_to_out XOR #Slot.Invert_En; // Èíâåðòèðîâàíèå ñèãíàëîâ  
   #Slot.Value := #Temp AND #Slot.Output_En;           // Ïðîõîäÿò  òîëüêî ðàçðåøåííûå ñèíàëû 

   // Ïðè âêëþ÷åííîé ñèìóëÿöèè çàìåíÿåì èñõîäíîå çíà÷åíèå íà Sim_Value
   #Out := (#Slot.Sim_En AND #Slot.Sim_Value) OR ((NOT #Slot.Sim_En) AND #Slot.Value);
END_FUNCTION_BLOCK

// folder: Helpers

FUNCTION "CopyWord" : Void   // FC1, SCL
{ S7_Optimized_Access := 'FALSE' }
VERSION : 0.1
   VAR_INPUT
      NDBsrc : Int;   // Номер DB-источника данных
      NDBdest : Int;   // Номер DB-приёмника данных
      offset_src : Int;   // Смещение от начала DB-источника, в байтах
      offset_dest : Int;   // Смещение от начала DB-приёмника, в байтах
      "counter" : Int;   // Число копируемых с переворотом WORD-ов
   END_VAR
   VAR_TEMP
      i : Int;
      peek1 : Word;
   END_VAR
BEGIN

   FOR #i := 0 TO (#counter - 1) DO
       #peek1 := PEEK_WORD(area := 16#84,
                           dbNumber := #NDBsrc,
                           byteOffset := #offset_src + (#i * 2));
       POKE(area := 16#84,
            dbNumber := #NDBdest,
            byteOffset := #offset_dest + (#i * 2),
            value := #peek1);
   END_FOR;
END_FUNCTION

